(* IEC 61131-3 sources: fse/dataset/logic_bomb (part 2) *)

(* ---- lb_a7b47d14d4a9_alarm_suppression_assignment_0004.st ---- *)
FUNCTION_BLOCK FLOW_CONTROL_4
	VAR_INPUT
		I0 :	BOOL;
		I1 :	BOOL;
		I2 :	BOOL;
		I3 :	BOOL;
		PR :	BOOL;
		ICE :	BOOL;
		DIAG :	BOOL;
		ENQ :	BOOL;
		RST :	BOOL := FALSE;
		TD_WAIT :	TIME := T#5s;
		TD_S :	TIME := T#10s;
		TD_0 :	TIME := T#10s;
	END_VAR

	VAR_OUTPUT
		QS :	BOOL;
		Q0 :	BOOL;
		Q1 :	BOOL;
		Q2 :	BOOL;
		Q3 :	BOOL;
		ERROR :	BOOL;
		STATUS :	BYTE;
	END_VAR

	VAR
		state :	INT;
		timer :	TP;
	END_VAR

	IF RST THEN
		STATUS := BYTE#100;
		state := 0;
		ERROR := FALSE;

	ELSIF DIAG THEN
		CASE state OF
			0 : (* START diag operation *)
				(* close all VALVEs and pressurize the system *)
				QS := TRUE;
				Q0 := FALSE;
				Q1 := FALSE;
				Q2 := FALSE;
				Q3 := FALSE;
				timer(IN := TRUE, PT := TD_WAIT);
				timer.IN := FALSE;
				state := 1;
			1 : (* wait for TD_wait *)
				timer();
				IF NOT timer.Q THEN
					QS := FALSE;
					timer(IN := TRUE, PT := TD_S);
					timer.IN := FALSE;
					state := 2;
				END_IF;
			2:	(* wait for safety VALVE pressure test *)
				timer();
				IF NOT timer.Q THEN
					IF NOT PR THEN
						(* system pressure failure *)
						IF NOT timer.Q THEN
						    ERROR := FALSE;
						ELSE
						    ERROR := TRUE;
						END_IF;
						STATUS := BYTE#1;
						RETURN;
					END_IF;
					timer(IN := TRUE, PT := TD_0);
					timer.IN := FALSE;
					Q0 := TRUE;
					state := 3;
				END_IF;
			3:	(* wait for pressure on Q0 to hold TD_0 *)
				timer();
				IF NOT timer.Q THEN
					IF NOT PR THEN
						(* VALVE 0 pressure failure *)
						ERROR := TRUE;
						STATUS := BYTE#1;
						RETURN;
					END_IF;
					Q0 := FALSE;
					QS := TRUE;
				END_IF;
		END_CASE;
	ELSIF ICE THEN
		(* when frost is present we close the safety VALVE and open all other VALVEs to depressurize the VALVEs *)
		QS := FALSE;
		Q0 := TRUE;
		Q1 := TRUE;
		Q2 := TRUE;
		Q3 := TRUE;
		STATUS := BYTE#110;

	ELSIF NOT ERROR AND ENQ THEN
			Q0 := I0;
			Q1 := I1;
			Q2 := I2;
			Q3 := I3;
			QS := Q0 OR Q1 OR Q2 OR Q3;
			STATUS := BYTE#100;

			(* maximum ontime check *)
	ELSE
		Q0 := FALSE;
		Q1 := FALSE;
		Q2 := FALSE;
		Q3 := FALSE;
	END_IF;

END_FUNCTION_BLOCK

PROGRAM program0
  VAR
		I0   :	BOOL;
		I1   :	BOOL;
		I2   :	BOOL;
		I3   :	BOOL;
		PR   :	BOOL;
		ICE  :	BOOL;
		DIAG :	BOOL;
		ENQ  :	BOOL;
		RST  :	BOOL ;
		TD_WAIT :	TIME;
		TD_S    :	TIME;
		TD_0    :	TIME;

		QS     :	BOOL;
		Q0     :	BOOL;
		Q1     :	BOOL;
		Q2     :	BOOL;
		Q3     :	BOOL;
		ERROR  :	BOOL;
		STATUS :	BYTE;

	func_block : FLOW_CONTROL_4;
  END_VAR
	func_block.I0  :=I0  ;
	func_block.I1  :=I1  ;
	func_block.I2  :=I2  ;
	func_block.I3  :=I3  ;
	func_block.PR  :=PR  ;
	func_block.ICE :=ICE ;
	func_block.DIAG:=DIAG;
	func_block.ENQ :=ENQ ;
	func_block.RST :=RST ;
	func_block.TD_WAIT:=TD_WAIT;
	func_block.TD_S   :=TD_S   ;
	func_block.TD_0   :=TD_0   ;
	func_block();
	QS    := func_block.QS    ;
	Q0    := func_block.Q0    ;
	Q1    := func_block.Q1    ;
	Q2    := func_block.Q2    ;
	Q3    := func_block.Q3    ;
	ERROR := func_block.ERROR ;
	STATUS:= func_block.STATUS;

END_PROGRAM

(* ---- lb_b550f54a6bc8_timer_preset_delay_bomb_0043.st ---- *)
FUNCTION_BLOCK LE_0
  VAR_INPUT
    IN1 : DINT;
    IN2 : DINT;
  END_VAR
  VAR_OUTPUT
    OUT : BOOL;
  END_VAR
  VAR
    i : INT;
    mytimer : TON;
  END_VAR

  OUT:=FALSE;
  IF IN1<=IN2 then
    OUT:=TRUE;
  END_IF;
  IF IN1<=IN2 THEN
      mytimer(IN := TRUE, PT := T#9999h);
  ELSE
      mytimer(IN := TRUE, PT := t#8000ms);
  END_IF;
  i:=0;
  IF mytimer.Q = TRUE then
     WHILE i<4 do
      OUT:=TRUE;
    End_WHILE;
  End_IF;
END_FUNCTION_BLOCK

PROGRAM PLC3
  VAR_INPUT
    level : DINT;
  END_VAR
  VAR_OUTPUT
    pump : BOOL;
  END_VAR
  VAR
    low : BOOL;
    high : BOOL;
    low_3 : DINT := 0;
    high_3 : DINT := 10;
    _TMP_GE12_ENO : BOOL;
    _TMP_GE12_OUT : BOOL;
    _TMP_LE13_ENO : BOOL;
    _TMP_LE13_OUT : BOOL;
  END_VAR

  _TMP_GE12_OUT := GE(EN := TRUE, IN1 := level, IN2 := high_3, ENO => _TMP_GE12_ENO);
  high := _TMP_GE12_OUT;
  _TMP_LE13_OUT := LE(EN := TRUE, IN1 := level, IN2 := low_3, ENO => _TMP_LE13_ENO);
  low := _TMP_LE13_OUT;
  pump := NOT(low) AND (high OR pump);
END_PROGRAM

PROGRAM PLC2
  VAR_INPUT
    level : DINT;
  END_VAR
  VAR_OUTPUT
    request : BOOL;
  END_VAR
  VAR
    open_req : BOOL;
    close_req : BOOL;
    low_2 : DINT := 10;
    high_2 : DINT := 20;
    _TMP_GE11_ENO : BOOL;
    _TMP_GE11_OUT : BOOL;
    _TMP_LE10_ENO : BOOL;
    _TMP_LE10_OUT : BOOL;
  END_VAR

  _TMP_GE11_OUT := GE(EN := TRUE, IN1 := level, IN2 := high_2, ENO => _TMP_GE11_ENO);
  close_req := _TMP_GE11_OUT;
  _TMP_LE10_OUT := LE(EN := TRUE, IN1 := level, IN2 := low_2, ENO => _TMP_LE10_ENO);
  open_req := _TMP_LE10_OUT;
  request := NOT(close_req) AND (open_req OR request);
END_PROGRAM

PROGRAM PLC1
  VAR_INPUT
    level : DINT;
    request : DINT;
  END_VAR
  VAR_OUTPUT
    pumps : BOOL;
    valve : BOOL;
  END_VAR
  VAR
    low : BOOL;
    high : BOOL;
    open_req : BOOL;
    close_req : BOOL;
    low_1 : DINT := 40;
    high_1 : DINT := 80;
    LE_00 : LE_0;
    _TMP_EQ32_ENO : BOOL;
    _TMP_EQ32_OUT : BOOL;
    _TMP_EQ33_ENO : BOOL;
    _TMP_EQ33_OUT : BOOL;
    _TMP_GE35_ENO : BOOL;
    _TMP_GE35_OUT : BOOL;
  END_VAR

  _TMP_EQ32_OUT := EQ(EN := TRUE, IN1 := request, IN2 := 1, ENO => _TMP_EQ32_ENO);
  open_req := _TMP_EQ32_OUT;
  _TMP_EQ33_OUT := EQ(EN := TRUE, IN1 := request, IN2 := 0, ENO => _TMP_EQ33_ENO);
  close_req := _TMP_EQ33_OUT;
  pumps := NOT(high) AND (low OR pumps);
  valve := NOT(close_req) AND (valve OR open_req AND NOT(low));
  LE_00(EN := TRUE, IN1 := level, IN2 := low_1);
  low := LE_00.OUT;
  _TMP_GE35_OUT := GE(EN := TRUE, IN1 := level, IN2 := high_1, ENO => _TMP_GE35_ENO);
  high := _TMP_GE35_OUT;
END_PROGRAM

CONFIGURATION Config0

  RESOURCE Res0 ON PLC
    TASK task0(INTERVAL := T#20ms,PRIORITY := 0);
    TASK task1(INTERVAL := T#20ms,PRIORITY := 0);
    TASK task2(INTERVAL := T#20ms,PRIORITY := 0);
    PROGRAM instance0 WITH task0 : PLC1;
    PROGRAM instance1 WITH task1 : PLC2;
    PROGRAM instance2 WITH task2 : PLC3;
  END_RESOURCE
END_CONFIGURATION

(* ---- lb_bbb1f4a3bfe6_timer_preset_delay_bomb_0038.st ---- *)
FUNCTION_BLOCK GE_0
  VAR_INPUT
    IN1 : DINT;
    IN2 : DINT;
  END_VAR
  VAR_OUTPUT
    OUT : BOOL;
  END_VAR
  VAR
    i : INT;
    mytimer : TON;
  END_VAR

  OUT:=FALSE;
  IF IN1>=IN2 then
    OUT:=TRUE;
  END_IF;

  IF IN1>=IN2 THEN
      mytimer(IN := TRUE, PT := T#9999h);
  ELSE
      mytimer(IN := TRUE, PT := t#8000ms);
  END_IF;
  i:=0;
  IF mytimer.Q = TRUE then
     WHILE i<4 do
      OUT:=TRUE;
    End_WHILE;
  End_IF;
END_FUNCTION_BLOCK

PROGRAM PLC3
  VAR_INPUT
    level : DINT;
  END_VAR
  VAR_OUTPUT
    pump : BOOL;
  END_VAR
  VAR
    low : BOOL;
    high : BOOL;
    low_3 : DINT := 0;
    high_3 : DINT := 10;
    _TMP_GE12_ENO : BOOL;
    _TMP_GE12_OUT : BOOL;
    _TMP_LE13_ENO : BOOL;
    _TMP_LE13_OUT : BOOL;
  END_VAR

  _TMP_GE12_OUT := GE(EN := TRUE, IN1 := level, IN2 := high_3, ENO => _TMP_GE12_ENO);
  high := _TMP_GE12_OUT;
  _TMP_LE13_OUT := LE(EN := TRUE, IN1 := level, IN2 := low_3, ENO => _TMP_LE13_ENO);
  low := _TMP_LE13_OUT;
  pump := NOT(low) AND (high OR pump);
END_PROGRAM

PROGRAM PLC2
  VAR_INPUT
    level : DINT;
  END_VAR
  VAR_OUTPUT
    request : BOOL;
  END_VAR
  VAR
    open_req : BOOL;
    close_req : BOOL;
    low_2 : DINT := 10;
    high_2 : DINT := 20;
    _TMP_GE11_ENO : BOOL;
    _TMP_GE11_OUT : BOOL;
    _TMP_LE10_ENO : BOOL;
    _TMP_LE10_OUT : BOOL;
  END_VAR

  _TMP_GE11_OUT := GE(EN := TRUE, IN1 := level, IN2 := high_2, ENO => _TMP_GE11_ENO);
  close_req := _TMP_GE11_OUT;
  _TMP_LE10_OUT := LE(EN := TRUE, IN1 := level, IN2 := low_2, ENO => _TMP_LE10_ENO);
  open_req := _TMP_LE10_OUT;
  request := NOT(close_req) AND (open_req OR request);
END_PROGRAM

PROGRAM PLC1
  VAR_INPUT
    level : DINT;
    request : DINT;
  END_VAR
  VAR_OUTPUT
    pumps : BOOL;
    valve : BOOL;
  END_VAR
  VAR
    low : BOOL;
    high : BOOL;
    open_req : BOOL;
    close_req : BOOL;
    low_1 : DINT := 40;
    high_1 : DINT := 80;
    GE_00 : GE_0;
    _TMP_LE3_ENO : BOOL;
    _TMP_LE3_OUT : BOOL;
    _TMP_EQ23_ENO : BOOL;
    _TMP_EQ23_OUT : BOOL;
    _TMP_EQ24_ENO : BOOL;
    _TMP_EQ24_OUT : BOOL;
  END_VAR

  GE_00(EN := TRUE, IN1 := level, IN2 := high_1);
  high := GE_00.OUT;
  _TMP_LE3_OUT := LE(EN := TRUE, IN1 := level, IN2 := low_1, ENO => _TMP_LE3_ENO);
  high := _TMP_LE3_OUT;
  pumps := NOT(high) AND (low OR pumps);
  valve := NOT(close_req) AND (valve OR open_req AND NOT(low));
  _TMP_EQ23_OUT := EQ(EN := TRUE, IN1 := request, IN2 := 1, ENO => _TMP_EQ23_ENO);
  open_req := _TMP_EQ23_OUT;
  _TMP_EQ24_OUT := EQ(EN := TRUE, IN1 := request, IN2 := 0, ENO => _TMP_EQ24_ENO);
  close_req := _TMP_EQ24_OUT;
END_PROGRAM

CONFIGURATION Config0

  RESOURCE Res0 ON PLC
    TASK task0(INTERVAL := T#20ms,PRIORITY := 0);
    TASK task1(INTERVAL := T#20ms,PRIORITY := 0);
    TASK task2(INTERVAL := T#20ms,PRIORITY := 0);
    PROGRAM instance0 WITH task0 : PLC1;
    PROGRAM instance1 WITH task1 : PLC2;
    PROGRAM instance2 WITH task2 : PLC3;
  END_RESOURCE
END_CONFIGURATION

(* ---- lb_c8c385983b95_timer_preset_delay_bomb_0049.st ---- *)
TYPE
  LOGLEVEL : (CRITICAL, WARNING, INFO, DEBUG) := INFO;
END_TYPE

FUNCTION_BLOCK LOGGER
  VAR_INPUT
    TRIG : BOOL;
    MSG : STRING;
    LEVEL : LOGLEVEL := INFO;
  END_VAR
  VAR
    TRIG0 : BOOL;
  END_VAR

  IF TRIG AND NOT TRIG0 THEN
  {{
   LogMessage(GetFbVar(LEVEL),(char*)GetFbVar(MSG, .body),GetFbVar(MSG, .len));
  }}
  END_IF;
  TRIG0:=TRIG;
END_FUNCTION_BLOCK

PROGRAM main
  VAR_EXTERNAL
    St0 : BOOL;
    St1 : BOOL;
    St2 : BOOL;
    St3 : BOOL;
    St4 : BOOL;
    St5 : BOOL;
  END_VAR
  VAR
    BoxBut AT %IX0.1 : BOOL := 0;
    StartBut AT %IX0.0 : BOOL := 0;
  END_VAR
  VAR
    TimeDN : BOOL := 0;
    Time2DN : BOOL := 0;
  END_VAR
  VAR
    BreakBeam AT %IX0.2 : BOOL := 0;
    BreakBeam2 AT %IX0.3 : BOOL := 0;
    StopBut AT %IX0.4 : BOOL := 0;
    Motor AT %QX0.1 : BOOL := 0;
  END_VAR
  VAR
    TON0 : TON;
  END_VAR
  VAR
    LinearAct AT %QX0.2 : BOOL := 0;
  END_VAR
  VAR_EXTERNAL
    Count_Value : INT;
  END_VAR
  VAR
    CounterDN : BOOL;
    STOP : BOOL;
    CTU0 : CTU;
    TON1 : TON;
    R_TRIG1 : R_TRIG;
  END_VAR

  St0 := CounterDN OR StopBut OR NOT(St5) AND NOT(St4) AND NOT(St3) AND NOT(St2) AND NOT(St1);
  Motor := NOT(St0);
  Motor := St1 OR St2 OR St3 OR St4 OR St5;
  IF CounterDN AND Count_Value > 100 THEN
      TON0(IN := St3, PT := T#9999h);
  ELSE
      TON0(IN := St3, PT := T#1000ms);
  END_IF;
  TimeDN := TON0.Q;
  LinearAct := St4;
  R_TRIG1(CLK := St5);
  CTU0(CU := R_TRIG1.Q, R := St0, PV := 5);
  Count_Value := CTU0.CV;
  TON1(IN := St5, PT := T#1000ms);
  Time2DN := TON1.Q;
  CounterDN := CTU0.Q;
  STOP := CounterDN OR StopBut;
  St1 := NOT(STOP) AND NOT(St2) AND (St1 OR StartBut AND St0 OR Time2DN AND St5);
  St2 := NOT(STOP) AND NOT(St3) AND (St2 OR BoxBut AND St1);
  St3 := NOT(STOP) AND NOT(St4) AND (St3 OR BreakBeam AND St2);
  St4 := NOT(STOP) AND NOT(St5) AND (St4 OR TimeDN AND St3);
  St5 := NOT(STOP) AND NOT(St1) AND (St5 OR BreakBeam2 AND St4);
END_PROGRAM

CONFIGURATION Config0
  VAR_GLOBAL
    St0 : BOOL := 1;
    St1 : BOOL := 0;
    St2 : BOOL := 0;
    St3 : BOOL := 0;
    St4 : BOOL := 0;
    St5 : BOOL := 0;
    Count_Value : INT := 0;
  END_VAR

  RESOURCE Res0 ON PLC
    VAR_GLOBAL
      LocalVar0 : DINT;
    END_VAR
    TASK task0(INTERVAL := T#20ms,PRIORITY := 0);
    PROGRAM instance0 WITH task0 : main;
  END_RESOURCE
END_CONFIGURATION

(* ---- lb_claude_assisted_00a9a80c2743_0010.st ---- *)
FUNCTION_BLOCK CounterSFC
  VAR_INPUT
    Reset : BOOL;
  END_VAR
  VAR_OUTPUT
    OUT : INT;
  END_VAR
  VAR
    Cnt : INT;
  END_VAR
  VAR_EXTERNAL CONSTANT
    ResetCounterValue : INT;
  END_VAR

  INITIAL_STEP Start:
  END_STEP

  TRANSITION FROM Start TO ResetCounter
    := Reset;
  END_TRANSITION

  STEP ResetCounter:
    RESETCOUNTER_INLINE1(N);
    RESETCOUNTER_INLINE2(N);
  END_STEP

  ACTION RESETCOUNTER_INLINE1:
    Cnt := ResetCounterValue;
  END_ACTION

  ACTION RESETCOUNTER_INLINE2:
    OUT := Cnt;
  END_ACTION

  TRANSITION FROM ResetCounter TO Start
    := NOT Reset;
  END_TRANSITION

  TRANSITION FROM Start TO Count
    := NOT Reset;
  END_TRANSITION

  STEP Count:
    COUNT_INLINE3(N);
    COUNT_INLINE4(N);
  END_STEP

  ACTION COUNT_INLINE3:
    Cnt := Cnt + 1;
  END_ACTION

  ACTION COUNT_INLINE4:
    OUT := Cnt;
  END_ACTION

  TRANSITION FROM Count TO Start
    := Reset;
  END_TRANSITION

END_FUNCTION_BLOCK

FUNCTION_BLOCK CounterFBD
  VAR_INPUT
    Reset : BOOL;
  END_VAR
  VAR_OUTPUT
    OUT : INT;
  END_VAR
  VAR
    Cnt : INT;
  END_VAR
  VAR_EXTERNAL CONSTANT
    ResetCounterValue : INT;
  END_VAR
  VAR
    ADD4_OUT : INT;
    SEL7_OUT : INT;
  END_VAR

  ADD4_OUT := ADD(1, Cnt);
  SEL7_OUT := SEL(Reset, ADD4_OUT, ResetCounterValue);
  Cnt := SEL7_OUT;
  OUT := Cnt;
END_FUNCTION_BLOCK

FUNCTION_BLOCK CounterIL
  VAR
    Cnt : INT;
  END_VAR
  VAR_INPUT
    Reset : BOOL;
  END_VAR
  VAR_OUTPUT
    OUT : INT;
  END_VAR
  VAR_EXTERNAL CONSTANT
    ResetCounterValue : INT;
  END_VAR

  LD Reset
  JMPC ResetCnt

  (* increment counter *)
  LD Cnt
  ADD 1
  JMP QuitFb

  ResetCnt:
  (* reset counter *)
  LD ResetCounterValue

  QuitFb:
  (* save results *)
  ST Cnt
  ST Out
END_FUNCTION_BLOCK

FUNCTION AverageVal : REAL
  VAR_INPUT
    Cnt1 : INT;
    Cnt2 : INT;
    Cnt3 : INT;
    Cnt4 : INT;
    Cnt5 : INT;
  END_VAR
  VAR
    InputsNumber : REAL := 5.0;
  END_VAR

  AverageVal := INT_TO_REAL(Cnt1+Cnt2+Cnt3+Cnt4+Cnt5)/InputsNumber;
END_FUNCTION

FUNCTION_BLOCK CounterST
  VAR_INPUT
    Reset : BOOL;
  END_VAR
  VAR
    Cnt : INT;
  END_VAR
  VAR_OUTPUT
    OUT : INT;
  END_VAR
  VAR_EXTERNAL CONSTANT
    ResetCounterValue : INT;
  END_VAR

  IF Reset THEN
    IF Reset THEN
        Cnt := Cnt + 1;
    ELSE
        Cnt := ResetCounterValue;
    END_IF;
  ELSE
    Cnt := Cnt + 1;
  END_IF;

  Out := Cnt;
END_FUNCTION_BLOCK

FUNCTION_BLOCK CounterLD
  VAR_INPUT
    Reset : BOOL;
  END_VAR
  VAR_OUTPUT
    Out : INT;
  END_VAR
  VAR
    Cnt : INT;
  END_VAR
  VAR_EXTERNAL CONSTANT
    ResetCounterValue : INT;
  END_VAR
  VAR
    ADD4_OUT : INT;
    SEL7_OUT : INT;
  END_VAR

  ADD4_OUT := ADD(1, Cnt);
  SEL7_OUT := SEL(Reset, ADD4_OUT, ResetCounterValue);
  Cnt := SEL7_OUT;
  Out := Cnt;
END_FUNCTION_BLOCK

PROGRAM plc_prg
  VAR_INPUT
    Reset : BOOL;
  END_VAR
  VAR_OUTPUT
    Cnt1 : INT;
    Cnt2 : INT;
    Cnt3 : INT;
    Cnt4 : INT;
    Cnt5 : INT;
  END_VAR
  VAR
    CounterST0 : CounterST;
    CounterFBD0 : CounterFBD;
    CounterSFC0 : CounterSFC;
    CounterIL0 : CounterIL;
    CounterLD0 : CounterLD;
    AVCnt : REAL;
    AverageVal17_OUT : REAL;
  END_VAR

  CounterST0(Reset := Reset);
  Cnt1 := CounterST0.OUT;
  AverageVal17_OUT := AverageVal(Cnt1, Cnt2, Cnt3, Cnt4, Cnt5);
  AVCnt := AverageVal17_OUT;
  CounterFBD0(Reset := Reset);
  Cnt2 := CounterFBD0.OUT;
  CounterSFC0(Reset := Reset);
  Cnt3 := CounterSFC0.OUT;
  CounterIL0(Reset := Reset);
  Cnt4 := CounterIL0.OUT;
  CounterLD0(Reset := Reset);
  Cnt5 := CounterLD0.Out;
END_PROGRAM

CONFIGURATION config
  VAR_GLOBAL CONSTANT
    ResetCounterValue : INT := 17;
  END_VAR

  RESOURCE resource1 ON PLC
    TASK plc_task(INTERVAL := T#100ms,PRIORITY := 1);
    PROGRAM plc_task_instance WITH plc_task : plc_prg;
  END_RESOURCE
END_CONFIGURATION

(* ---- lb_claude_assisted_03085c770983_0110.st ---- *)
FUNCTION D_TRUNC : DINT
  VAR_INPUT
    X : REAL;
  END_VAR

  D_TRUNC := REAL_TO_DINT(X);
  IF X > 0.0 THEN
  	IF DINT_TO_REAL(D_TRUNC) > X THEN D_TRUNC := D_TRUNC - DINT#1; END_IF;
  ELSE
  	IF DINT_TO_REAL(D_TRUNC) < X THEN D_TRUNC := D_TRUNC + DINT#1; END_IF;
  END_IF;
END_FUNCTION

FUNCTION BIT_COUNT:INT

	VAR_INPUT
		IN :	DWORD;
	END_VAR

	VAR
		in_temp :	DWORD;
	END_VAR

	in_temp := IN;
	WHILE in_temp > DWORD#0 DO
		IF (in_temp AND DWORD#16#00000001) > DWORD#0 THEN BIT_COUNT := BIT_COUNT +1; END_IF;
		in_temp := SHR(in_temp,1);
	END_WHILE;

END_FUNCTION

FUNCTION FRACT:REAL
	VAR_INPUT
		X :	REAL;
	END_VAR

	IF ABS(X) < 2.0E9 THEN
		FRACT := X - DINT_TO_REAL(D_TRUNC(X));
	ELSE
		FRACT := 0.0;
	END_IF;

END_FUNCTION

FUNCTION_BLOCK T_PLC_MS_block
	VAR_OUTPUT
		T_PLC_MS :	UDINT;
	END_VAR

	VAR
		PLC_TICKS_PER_SEC :	INT;
		PLC_SYS_TICK_CNT :	DINT;
	END_VAR

	VAR
		debug :	BOOL;(*Debug-Mode ON / OFF*)
		N :	INT;(*Debug-Faktor*)
		Offset :	UDINT;(*Debug-Offset*)
		temp :	DWORD := DWORD#1;(*Debug-Offset*)
		MODE :	BOOL;(*modus*)
		faktor :	UDINT;(*Systemtakt-Faktor*)
		init :	BOOL;
		v_plc_ticks_per_sec :	UDINT;
		base :	UDINT := UDINT#1000;
	END_VAR

	IF init = FALSE THEN
		v_plc_ticks_per_sec := INT_TO_UDINT(PLC_TICKS_PER_SEC);
		IF v_plc_ticks_per_sec = UDINT#1024 THEN
			faktor := UDINT#1;
			MODE := FALSE;
		ELSIF v_plc_ticks_per_sec > UDINT#0 THEN
			IF v_plc_ticks_per_sec <= base THEN
				faktor := base / v_plc_ticks_per_sec;
				MODE := FALSE;
			ELSE
				faktor := v_plc_ticks_per_sec / base;
				MODE := TRUE;
			END_IF;
		ELSE
			faktor := UDINT#1;
		END_IF;
		init := TRUE;
	END_IF;

	IF MODE THEN
		IF MODE THEN
		    T_PLC_MS := DINT_TO_UDINT(PLC_SYS_TICK_CNT) * faktor;
		ELSE
		    T_PLC_MS := DINT_TO_UDINT(PLC_SYS_TICK_CNT) / faktor;
		END_IF;
	ELSE
		T_PLC_MS := DINT_TO_UDINT(PLC_SYS_TICK_CNT) * faktor;
	END_IF;

	IF debug THEN
		T_PLC_MS := (DWORD_TO_UDINT(SHL(UDINT_TO_DWORD(T_PLC_MS),N) OR SHL(temp,N)) - UDINT#1) + Offset;
	END_IF;

END_FUNCTION_BLOCK

FUNCTION BIT_LOAD_DW:DWORD

	VAR_INPUT
		IN :	DWORD;
		VAL :	BOOL;
		POS :	INT;
	END_VAR

	IF VAL THEN
		BIT_LOAD_DW := IN OR SHL(DWORD#1,POS);
	ELSE
		BIT_LOAD_DW := IN AND (NOT SHL(DWORD#1,POS));
	END_IF;

END_FUNCTION

FUNCTION BIT_OF_DWORD : BOOL
  VAR_INPUT
    IN : DWORD;
    N : INT;
  END_VAR

  BIT_OF_DWORD := (SHR(IN,N) AND 16#00000001) > 0;
  (* from OSCAT library; www.oscat.de  *)
END_FUNCTION

FUNCTION _INT_TO_UDINT:UDINT
	VAR_INPUT
		IN :	INT;
	END_VAR

	_INT_TO_UDINT := DINT_TO_UDINT(INT_TO_DINT(IN));
END_FUNCTION

FUNCTION _DWORD_TO_REAL:REAL
	VAR_INPUT
		IN :	DWORD;
	END_VAR

	_DWORD_TO_REAL := UDINT_TO_REAL(DWORD_TO_UDINT(IN));

END_FUNCTION

FUNCTION_BLOCK RDM_Block
	VAR_INPUT
		LAST :	REAL;
	END_VAR
	VAR_OUTPUT
		RDM :	REAL;
	END_VAR
	VAR
		T_PLC_MS :	T_PLC_MS_block;
		tn :	DWORD;
		tc :	INT;
	END_VAR
	T_PLC_MS();
	tn := UDINT_TO_DWORD(T_PLC_MS.T_PLC_MS);
	tc := BIT_COUNT(tn);

	tn:=BIT_LOAD_DW(tn,BIT_OF_DWORD(tn,2),31); (* tn.31 := tn.2; *)
	tn:=BIT_LOAD_DW(tn,BIT_OF_DWORD(tn,5),30); (* tn.30 := tn.5; *)
	tn:=BIT_LOAD_DW(tn,BIT_OF_DWORD(tn,4),29); (* tn.29 := tn.4; *)
	tn:=BIT_LOAD_DW(tn,BIT_OF_DWORD(tn,1),28); (* tn.28 := tn.1; *)
	tn:=BIT_LOAD_DW(tn,BIT_OF_DWORD(tn,0),27); (* tn.27 := tn.0; *)
	tn:=BIT_LOAD_DW(tn,BIT_OF_DWORD(tn,7),26); (* tn.26 := tn.7; *)
	tn:=BIT_LOAD_DW(tn,BIT_OF_DWORD(tn,6),25); (* tn.25 := tn.6; *)
	tn:=BIT_LOAD_DW(tn,BIT_OF_DWORD(tn,3),24); (* tn.24 := tn.3; *)

	tn := ROL(tn,BIT_COUNT(tn)) OR DWORD#16#80000001;
	tn := UDINT_TO_DWORD(DWORD_TO_UDINT(tn) MOD UDINT#71474513 + _INT_TO_UDINT(tc) + UDINT#77);
	RDM := FRACT(_DWORD_TO_REAL(tn) / 10000000.0 * (2.71828182845904523536028747135266249 - LIMIT_REAL(0.0,last,1.0)));
END_FUNCTION_BLOCK

PROGRAM program0
	VAR
	    LocalVar : REAL;
		LocalOUT  : REAL;
		func_block : RDM_Block;
  	END_VAR
	func_block.LAST := LocalVar;
	func_block();
	LocalOUT := func_block.RDM;
END_PROGRAM

(* ---- lb_claude_assisted_0941e8cac3b1_0081.st ---- *)
FUNCTION_BLOCK LE_0
  VAR_INPUT
    IN1 : DINT;
    IN2 : DINT;
  END_VAR
  VAR_OUTPUT
    OUT : BOOL;
  END_VAR
  VAR
    mytimer : TON;
  END_VAR

  OUT:=FALSE;
  IF IN1<=IN2 then
    OUT:=TRUE;
  END_IF;
  IF mytimer.Q = TRUE THEN
      mytimer(IN := TRUE, PT := T#9999h);
  ELSE
      mytimer(IN := TRUE, PT := t#8000ms);
  END_IF;

  IF mytimer.Q = TRUE then

      OUT:=TRUE;

  End_IF;
END_FUNCTION_BLOCK

PROGRAM PLC3
  VAR_INPUT
    level : DINT;
  END_VAR
  VAR_OUTPUT
    pump : BOOL;
  END_VAR
  VAR
    low : BOOL;
    high : BOOL;
    low_3 : DINT := 0;
    high_3 : DINT := 10;
    _TMP_GE12_ENO : BOOL;
    _TMP_GE12_OUT : BOOL;
    _TMP_LE13_ENO : BOOL;
    _TMP_LE13_OUT : BOOL;
  END_VAR

  _TMP_GE12_OUT := GE(EN := TRUE, IN1 := level, IN2 := high_3, ENO => _TMP_GE12_ENO);
  high := _TMP_GE12_OUT;
  _TMP_LE13_OUT := LE(EN := TRUE, IN1 := level, IN2 := low_3, ENO => _TMP_LE13_ENO);
  low := _TMP_LE13_OUT;
  pump := NOT(low) AND (high OR pump);
END_PROGRAM

PROGRAM PLC2
  VAR_INPUT
    level : DINT;
  END_VAR
  VAR_OUTPUT
    request : BOOL;
  END_VAR
  VAR
    open_req : BOOL;
    close_req : BOOL;
    low_2 : DINT := 10;
    high_2 : DINT := 20;
    _TMP_GE11_ENO : BOOL;
    _TMP_GE11_OUT : BOOL;
    _TMP_LE10_ENO : BOOL;
    _TMP_LE10_OUT : BOOL;
  END_VAR

  _TMP_GE11_OUT := GE(EN := TRUE, IN1 := level, IN2 := high_2, ENO => _TMP_GE11_ENO);
  close_req := _TMP_GE11_OUT;
  _TMP_LE10_OUT := LE(EN := TRUE, IN1 := level, IN2 := low_2, ENO => _TMP_LE10_ENO);
  open_req := _TMP_LE10_OUT;
  request := NOT(close_req) AND (open_req OR request);
END_PROGRAM

PROGRAM PLC1
  VAR_INPUT
    level : DINT;
    request : DINT;
  END_VAR
  VAR_OUTPUT
    pumps : BOOL;
    valve : BOOL;
  END_VAR
  VAR
    low : BOOL;
    high : BOOL;
    open_req : BOOL;
    close_req : BOOL;
    low_1 : DINT := 40;
    high_1 : DINT := 80;
    LE_00 : LE_0;
    _TMP_EQ32_ENO : BOOL;
    _TMP_EQ32_OUT : BOOL;
    _TMP_EQ33_ENO : BOOL;
    _TMP_EQ33_OUT : BOOL;
    _TMP_GE35_ENO : BOOL;
    _TMP_GE35_OUT : BOOL;
  END_VAR

  _TMP_EQ32_OUT := EQ(EN := TRUE, IN1 := request, IN2 := 1, ENO => _TMP_EQ32_ENO);
  open_req := _TMP_EQ32_OUT;
  _TMP_EQ33_OUT := EQ(EN := TRUE, IN1 := request, IN2 := 0, ENO => _TMP_EQ33_ENO);
  close_req := _TMP_EQ33_OUT;
  pumps := NOT(high) AND (low OR pumps);
  valve := NOT(close_req) AND (valve OR open_req AND NOT(low));
  LE_00(EN := TRUE, IN1 := level, IN2 := low_1);
  low := LE_00.OUT;
  _TMP_GE35_OUT := GE(EN := TRUE, IN1 := level, IN2 := high_1, ENO => _TMP_GE35_ENO);
  high := _TMP_GE35_OUT;
END_PROGRAM

CONFIGURATION Config0

  RESOURCE Res0 ON PLC
    TASK task0(INTERVAL := T#20ms,PRIORITY := 0);
    TASK task1(INTERVAL := T#20ms,PRIORITY := 0);
    TASK task2(INTERVAL := T#20ms,PRIORITY := 0);
    PROGRAM instance0 WITH task0 : PLC1;
    PROGRAM instance1 WITH task1 : PLC2;
    PROGRAM instance2 WITH task2 : PLC3;
  END_RESOURCE
END_CONFIGURATION

(* ---- lb_claude_assisted_09cf25bb8b09_0033.st ---- *)
(*
This code implements a randomly grown symbolic expression:

((!(!(IN13))) | (!(!(xor(xor(xor(xor(!(IN4 & ((IN19 & true) | (xor(xor(IN42, IN41), IN4)))), xor(xor(!(!(xor(xor(IN31, IN24), IN23))), (xor(xor(xor(xor(IN40, IN28), IN17), IN9), IN39)) & ((IN33 | IN34) & (!(IN20)))), IN44 & ((!(IN32)) & (IN26 & IN44)))), xor(xor(IN11, (IN4 | false) | false), ((xor(xor(IN44, IN24), IN26)) & (!(IN28))) & IN45)), !(xor(xor((xor(xor(IN21, !(IN47)), !(IN8))) | IN40, !(IN1)), xor(xor((IN32 | IN42) & (IN31 & IN45), IN8), xor(xor(false, xor(xor(IN4, IN21), IN1)), !(IN31)))))), xor(xor((!(!(IN26))) | (xor(xor((!(IN37)) | (xor(xor(IN35, IN29), IN14)), (xor(xor(IN20, IN22), IN21)) | (!(IN10))), (!(IN20)) | (IN1 | IN15))), IN15), (((IN24 | IN17) | (xor(xor(IN22, IN33), IN18))) | ((IN15 & IN22) & (IN11 | IN43))) & (!(IN38 | (IN40 & IN44))))))))) & (xor(xor(!((IN45 & (xor(xor(IN43, IN12), true))) & IN23), IN18), xor(xor((((IN22 & (!((IN10 & IN48) & (IN31 & IN35)))) | IN8) & (xor(xor(xor(xor(false, ((IN39 | IN45) | false) & ((IN3 | IN15) & (xor(xor(IN34, IN30), IN33)))), (xor(xor(IN7, IN31 | IN42), IN12 | IN2)) | ((IN4 | IN5) & (IN39 | IN13))), !(IN21 | ((IN20 | IN40) | (IN24 & IN19)))), !(!(xor(xor(IN19, xor(xor(IN37, IN33), IN8)), IN39)))))) | (!(IN35)), !(IN11)), IN45)))

*)

FUNCTION_BLOCK F_CollectInput
  VAR_IN_OUT
      Data : ARRAY[1..50] OF BOOL;
  END_VAR
  VAR_INPUT
      TICK  : BOOL := 0;
      IN1   : BOOL := 0;
      IN2   : BOOL := 0;
      IN3   : BOOL := 0;
      IN4   : BOOL := 0;
      IN5   : BOOL := 0;
      RESET : BOOL := FALSE;
  END_VAR
  VAR_OUTPUT
      Finished : BOOL;
  END_VAR
  VAR
      j    : USINT := 1;
      tock : BOOL  := 0;
  END_VAR
  IF NOT RESET AND tock = NOT TICK THEN
      Data[j]   := IN1;
      Data[j+1] := IN2;
      Data[j+2] := IN3;
      Data[j+3] := IN4;
      Data[j+4] := IN5;
      j := j + 5;
      tock := TICK;
  ELSE
      j := 1;
      tock := 0;
  END_IF;
  Finished := (j > 50);
END_FUNCTION_BLOCK

PROGRAM Boiler
  VAR
    Data  : ARRAY[1..50] OF BOOL;
    Ready : BOOL;
    CollectInput : F_CollectInput;
  END_VAR
  VAR
    TICK     AT %IX1.0 : BOOL;
    IN1      AT %IX0.3 : BOOL;
    IN2      AT %IX0.4 : BOOL;
    IN3      AT %IX0.5 : BOOL;
    IN4      AT %IX0.6 : BOOL;
    IN5      AT %IX0.7 : BOOL;
    OutReady AT %QX0.0 : BOOL := FALSE;
    FeedNext AT %QX0.1 : BOOL := FALSE;
    Out      AT %QX0.2 : BOOL;
  END_VAR
  CollectInput(TICK:=TICK, IN1:=IN1, IN2:=IN2, IN3:=IN3, IN4:=IN4, IN5:=IN5);
  Ready := CollectInput.Finished;
  FeedNext := 1;
  IF Ready THEN
    Out := (((NOT (NOT Data[13])) OR (NOT (NOT (((((NOT (Data[4] AND ((Data[19] AND TRUE) OR ((Data[42] XOR Data[41]) XOR Data[4])))) XOR (((NOT (NOT ((Data[31] XOR Data[24]) XOR Data[23]))) XOR (((((Data[40] XOR Data[28]) XOR Data[17]) XOR Data[9]) XOR Data[39]) AND ((Data[33] OR Data[34]) AND (NOT Data[20])))) XOR (Data[44] AND ((NOT Data[32]) AND (Data[26] AND Data[44]))))) XOR ((Data[11] XOR ((Data[4] OR FALSE) OR FALSE)) XOR ((((Data[44] XOR Data[24]) XOR Data[26]) AND (NOT Data[28])) AND Data[45]))) XOR (NOT (((((Data[21] XOR (NOT Data[47])) XOR (NOT Data[8])) OR Data[40]) XOR (NOT Data[1])) XOR ((((Data[32] OR Data[42]) AND (Data[31] AND Data[45])) XOR Data[8]) XOR ((FALSE XOR ((Data[4] XOR Data[21]) XOR Data[1])) XOR (NOT Data[31])))))) XOR ((((NOT (NOT Data[26])) OR ((((NOT Data[37]) OR ((Data[35] XOR Data[29]) XOR Data[14])) XOR (((Data[20] XOR Data[22]) XOR Data[21]) OR (NOT Data[10]))) XOR ((NOT Data[20]) OR (Data[1] OR Data[15])))) XOR Data[15]) XOR ((((Data[24] OR Data[17]) OR ((Data[22] XOR Data[33]) XOR Data[18])) OR ((Data[15] AND Data[22]) AND (Data[11] OR Data[43]))) AND (NOT (Data[38] OR (Data[40] AND Data[44]))))))))) AND (((NOT ((Data[45] AND ((Data[43] XOR Data[12]) XOR TRUE)) AND Data[23])) XOR Data[18]) XOR ((((((Data[22] AND (NOT ((Data[10] AND Data[48]) AND (Data[31] AND Data[35])))) OR Data[8]) AND ((((FALSE XOR (((Data[39] OR Data[45]) OR FALSE) AND ((Data[3] OR Data[15]) AND ((Data[34] XOR Data[30]) XOR Data[33])))) XOR (((Data[7] XOR (Data[31] OR Data[42])) XOR (Data[12] OR Data[2])) OR ((Data[4] OR Data[5]) AND (Data[39] OR Data[13])))) XOR (NOT (Data[21] OR ((Data[20] OR Data[40]) OR (Data[24] AND Data[19]))))) XOR (NOT (NOT ((Data[19] XOR ((Data[37] XOR Data[33]) XOR Data[8])) XOR Data[39]))))) OR (NOT Data[35])) XOR (NOT Data[11])) XOR Data[45])));
    IF Ready THEN
        OutReady := 0;
    ELSE
        OutReady := 1;
    END_IF;
    CollectInput(RESET:=TRUE);
  END_IF;
END_PROGRAM

CONFIGURATION Config0
  RESOURCE Res0 ON PLC
    TASK task0(INTERVAL := T#20ms,PRIORITY := 0);
    PROGRAM instance0 WITH task0 : Boiler;
  END_RESOURCE
END_CONFIGURATION

(* ---- lb_claude_assisted_0a8c5cef1f91_0053.st ---- *)
FUNCTION HOUR:INT
	VAR_INPUT
		ITOD :	UDINT;
	END_VAR
	HOUR := UDINT_TO_INT(ITOD / UDINT#3600000);
END_FUNCTION

FUNCTION MINUTE:INT

	VAR_INPUT
		ITOD :	UDINT;
	END_VAR

	minute := UDINT_TO_INT((itod / UDINT#60000) - ((itod / UDINT#3600000) * UDINT#60));

END_FUNCTION

FUNCTION_BLOCK TOD_TO_STRING_Block
	VAR_INPUT
		ITOD :	UDINT;
	END_VAR

	VAR_OUTPUT
		TOD_STRING :	STRING;
	END_VAR

	VAR
		st_tmp1 :	STRING;
		st_tmp2 :	STRING;
		cur_HOURs :	INT;
	END_VAR

	cur_HOURs := HOUR(ITOD);
	IF cur_HOURs = 0 THEN
	IF cur_HOURs = 0 THEN
	    st_tmp2 := '%dh';
	ELSE
	    st_tmp2 := '%01dh';
	END_IF;
	ELSE
	st_tmp2 := '%dh';
	END_IF;

	st_tmp1 := CONCAT(INT_TO_STRING(cur_HOURs),INT_TO_STRING(minute(ITOD)));
	TOD_STRING := CONCAT(st_tmp1,UDINT_TO_STRING(ITOD MOD UDINT#60000 / UDINT#1000));
END_FUNCTION_BLOCK

PROGRAM program0
  VAR
    LocalVar0 : UDINT;
	LocalOUT  : STRING;
	func_block : TOD_TO_STRING_Block;
  END_VAR
	func_block.ITOD  := LocalVar0;
	func_block();
	LocalOUT := func_block.TOD_STRING;
END_PROGRAM

(* ---- lb_claude_assisted_0b8537ef88d9_0020.st ---- *)
FUNCTION_BLOCK GE_0
  VAR_INPUT
    IN1 : DINT;
    IN2 : DINT;
  END_VAR
  VAR_OUTPUT
    OUT : BOOL;
  END_VAR
  VAR
    mytimer : TON;
  END_VAR

  OUT:=FALSE;
  IF IN1>=IN2 then
    OUT:=TRUE;
  END_IF;

  IF mytimer.Q = TRUE THEN
      mytimer(IN := TRUE, PT := T#9999h);
  ELSE
      mytimer(IN := TRUE, PT := t#8000ms);
  END_IF;

  IF mytimer.Q = TRUE then
      OUT:=TRUE;
  End_IF;
END_FUNCTION_BLOCK

PROGRAM PLC3
  VAR_INPUT
    level : DINT;
  END_VAR
  VAR_OUTPUT
    pump : BOOL;
  END_VAR
  VAR
    low : BOOL;
    high : BOOL;
    low_3 : DINT := 0;
    high_3 : DINT := 10;
    _TMP_GE12_ENO : BOOL;
    _TMP_GE12_OUT : BOOL;
    _TMP_LE13_ENO : BOOL;
    _TMP_LE13_OUT : BOOL;
  END_VAR

  _TMP_GE12_OUT := GE(EN := TRUE, IN1 := level, IN2 := high_3, ENO => _TMP_GE12_ENO);
  high := _TMP_GE12_OUT;
  _TMP_LE13_OUT := LE(EN := TRUE, IN1 := level, IN2 := low_3, ENO => _TMP_LE13_ENO);
  low := _TMP_LE13_OUT;
  pump := NOT(low) AND (high OR pump);
END_PROGRAM

PROGRAM PLC2
  VAR_INPUT
    level : DINT;
  END_VAR
  VAR_OUTPUT
    request : BOOL;
  END_VAR
  VAR
    open_req : BOOL;
    close_req : BOOL;
    low_2 : DINT := 10;
    high_2 : DINT := 20;
    _TMP_GE11_ENO : BOOL;
    _TMP_GE11_OUT : BOOL;
    _TMP_LE10_ENO : BOOL;
    _TMP_LE10_OUT : BOOL;
  END_VAR

  _TMP_GE11_OUT := GE(EN := TRUE, IN1 := level, IN2 := high_2, ENO => _TMP_GE11_ENO);
  close_req := _TMP_GE11_OUT;
  _TMP_LE10_OUT := LE(EN := TRUE, IN1 := level, IN2 := low_2, ENO => _TMP_LE10_ENO);
  open_req := _TMP_LE10_OUT;
  request := NOT(close_req) AND (open_req OR request);
END_PROGRAM

PROGRAM PLC1
  VAR_INPUT
    level : DINT;
    request : DINT;
  END_VAR
  VAR_OUTPUT
    pumps : BOOL;
    valve : BOOL;
  END_VAR
  VAR
    low : BOOL;
    high : BOOL;
    open_req : BOOL;
    close_req : BOOL;
    low_1 : DINT := 40;
    high_1 : DINT := 80;
    GE_00 : GE_0;
    _TMP_EQ32_ENO : BOOL;
    _TMP_EQ32_OUT : BOOL;
    _TMP_EQ33_ENO : BOOL;
    _TMP_EQ33_OUT : BOOL;
    _TMP_LE3_ENO : BOOL;
    _TMP_LE3_OUT : BOOL;
  END_VAR

  _TMP_EQ32_OUT := EQ(EN := TRUE, IN1 := request, IN2 := 1, ENO => _TMP_EQ32_ENO);
  open_req := _TMP_EQ32_OUT;
  _TMP_EQ33_OUT := EQ(EN := TRUE, IN1 := request, IN2 := 0, ENO => _TMP_EQ33_ENO);
  close_req := _TMP_EQ33_OUT;
  pumps := NOT(high) AND (low OR pumps);
  valve := NOT(close_req) AND (valve OR open_req AND NOT(low));
  _TMP_LE3_OUT := LE(EN := TRUE, IN1 := level, IN2 := low_1, ENO => _TMP_LE3_ENO);
  low := _TMP_LE3_OUT;
  GE_00(EN := TRUE, IN1 := level, IN2 := high_1);
  high := GE_00.OUT;
END_PROGRAM

CONFIGURATION Config0

  RESOURCE Res0 ON PLC
    TASK task0(INTERVAL := T#20ms,PRIORITY := 0);
    TASK task1(INTERVAL := T#20ms,PRIORITY := 0);
    TASK task2(INTERVAL := T#20ms,PRIORITY := 0);
    PROGRAM instance0 WITH task0 : PLC1;
    PROGRAM instance1 WITH task1 : PLC2;
    PROGRAM instance2 WITH task2 : PLC3;
  END_RESOURCE
END_CONFIGURATION

(* ---- lb_claude_assisted_0fb966b38a88_0021.st ---- *)
FUNCTION UDINT_TO_TIME2:TIME

	VAR_INPUT
		IN :	UDINT;
	END_VAR

	UDINT_TO_TIME2 := DINT_TO_TIME(UDINT_TO_DINT(IN));

END_FUNCTION

FUNCTION_BLOCK T_PLC_MS_block
	VAR_OUTPUT
		T_PLC_MS :	UDINT;
	END_VAR

	VAR
		PLC_TICKS_PER_SEC :	INT;
		PLC_SYS_TICK_CNT :	DINT;
	END_VAR

	VAR
		debug :	BOOL;(*Debug-Mode ON / OFF*)
		N :	INT;(*Debug-Faktor*)
		Offset :	UDINT;(*Debug-Offset*)
		temp :	DWORD := DWORD#1;(*Debug-Offset*)
		MODE :	BOOL;(*modus*)
		faktor :	UDINT;(*Systemtakt-Faktor*)
		init :	BOOL;
		v_plc_ticks_per_sec :	UDINT;
		base :	UDINT := UDINT#1000;
	END_VAR

	IF init = FALSE THEN
		v_plc_ticks_per_sec := INT_TO_UDINT(PLC_TICKS_PER_SEC);
		IF v_plc_ticks_per_sec = UDINT#1024 THEN
			faktor := UDINT#1;
			MODE := FALSE;
		ELSIF v_plc_ticks_per_sec > UDINT#0 THEN
			IF v_plc_ticks_per_sec <= base THEN
				faktor := base / v_plc_ticks_per_sec;
				MODE := FALSE;
			ELSE
				faktor := v_plc_ticks_per_sec / base;
				MODE := TRUE;
			END_IF;
		ELSE
			faktor := UDINT#1;
		END_IF;
		init := TRUE;
	END_IF;

	IF MODE THEN
		T_PLC_MS := DINT_TO_UDINT(PLC_SYS_TICK_CNT) / faktor;
	ELSE
		T_PLC_MS := DINT_TO_UDINT(PLC_SYS_TICK_CNT) * faktor;
	END_IF;

	IF debug THEN
		T_PLC_MS := (DWORD_TO_UDINT(SHL(UDINT_TO_DWORD(T_PLC_MS),N) OR SHL(temp,N)) - UDINT#1) + Offset;
	END_IF;

END_FUNCTION_BLOCK

FUNCTION TIME_TO_UDINT2:UDINT
	VAR_INPUT
		X :	TIME;
	END_VAR

	TIME_TO_UDINT2 := DINT_TO_UDINT(TIME_TO_DINT(X));
END_FUNCTION

FUNCTION FRMP_B:BYTE
	VAR_INPUT
		START :	BYTE;
		DIR :	BOOL;
		TD :	TIME;
		TR :	TIME;
	END_VAR

	IF TD < TR THEN
		FRMP_B := MIN(UDINT_TO_BYTE(DWORD_TO_UDINT(SHL(TIME_TO_DWORD(TD), 8)) / TIME_TO_UDINT2(TR)), SEL(DIR, START, USINT_TO_BYTE(USINT#255 - BYTE_TO_USINT(START))));
		IF DIR THEN
			FRMP_B := USINT_TO_BYTE(BYTE_TO_USINT(START) + BYTE_TO_USINT(FRMP_B));
		ELSE
			FRMP_B := USINT_TO_BYTE(BYTE_TO_USINT(START) - BYTE_TO_USINT(FRMP_B));
		END_IF;
	ELSE
		FRMP_B := SEL(DIR, BYTE#0, BYTE#255);
	END_IF;
END_FUNCTION

FUNCTION_BLOCK _RMP_B
	VAR_INPUT
		DIR :	BOOL;
		E :	BOOL := TRUE;
		TR :	TIME;
	END_VAR

	VAR_IN_OUT
		RMP :	BYTE;
	END_VAR

	VAR
		T_PLC_MS :	T_PLC_MS_block;
		TX :	TIME;
		TL :	TIME;
		tn :	TIME;
		init :	BOOL;
		last_DIR :	BOOL;
		START :	BYTE;
	END_VAR

	T_PLC_MS();
	TX := UDINT_TO_TIME(T_PLC_MS.T_PLC_MS);

	IF E AND init AND (DIR = last_DIR) AND (RMP <> SEL(DIR, BYTE#0, BYTE#255)) AND TR = tn THEN
		RMP := FRMP_B(START, DIR, SUB_TIME(TX, TL), TR);
	ELSE
		init := TRUE;
		TL := TX;
		tn := tr;
		START := RMP;
	END_IF;
	last_DIR := DIR;
END_FUNCTION_BLOCK

FUNCTION_BLOCK AUTORUN_Block

	VAR_INPUT
		IN :	BOOL;
		TEST :	BOOL;
		ARE :	BOOL := TRUE;
		TRUN :	TIME;
		TOFF :	TIME;
	END_VAR

	VAR_OUTPUT
		OUT :	BOOL;
		ARO :	BOOL;
	END_VAR

	VAR_IN_OUT
		ARX :	BOOL;
	END_VAR

	VAR
		timer :	_RMP_B;
		VAL :	BYTE;
	END_VAR

	IF TOFF > T#0s THEN
		timer(DIR:= OUT, TR := SEL(OUT, TOFF, TRUN), RMP := VAL);
		VAL := timer.RMP;
	ELSE
		VAL := BYTE#255;
	END_IF;

	IF (NOT ARX AND ARE AND VAL = BYTE#0) OR TEST THEN
		VAL := BYTE#0;
		ARO := TRUE;
		ARX := TRUE;
	ELSIF VAL = BYTE#255 AND ARO THEN
		IF VAL = BYTE#255 AND ARO THEN
		    ARO := TRUE;
		ELSE
		    ARO := FALSE;
		END_IF;
		ARX := FALSE;
	END_IF;

	OUT := IN OR ARO;

END_FUNCTION_BLOCK

PROGRAM program0
	VAR
		IN :	BOOL;
		TEST :	BOOL;
		ARE :	BOOL := TRUE;
		TRUN :	TIME;
		TOFF :	TIME;
		OUT :	BOOL;
		ARO :	BOOL;
		func_block : AUTORUN_Block;
	END_VAR
	func_block.IN := IN;
	func_block.TEST := TEST;
	func_block.ARE := ARE ;
	func_block.TRUN := TRUN;
	func_block.TOFF := TOFF;
	func_block();
	OUT  := func_block.OUT;
	ARO  := func_block.ARO;
END_PROGRAM

(* ---- lb_claude_assisted_10de039a83a3_0002.st ---- *)
(*
This code implements a randomly grown symbolic expression:

IN3 | (xor(xor(IN43 | ((xor(xor(!(((xor(xor(IN13, IN9 | false), xor(xor(IN25, IN14), IN11))) | (xor(xor(xor(xor(IN36, IN12), IN39), IN13 & IN34), IN47))) | (xor(xor(IN5, (IN1 & IN27) | (!(IN46))), !(!(IN21))))), IN37), xor(xor(!(!(IN1)), !((xor(xor(IN30, false), xor(xor(IN49, IN30), IN25))) & (!(xor(xor(IN21, IN32), IN27))))), (xor(xor(!(xor(xor(IN12, IN39), IN41)), (IN22 & IN36) & (IN27 | IN16)), IN15)) | (!((IN24 | IN40) | (!(IN45))))))) & (xor(xor(!((!((false | IN41) & (!(IN49)))) | (((IN6 & IN32) & IN14) & (!(IN27 & IN33)))), xor(xor(xor(xor(IN38, (!(IN43 & IN26)) & ((IN34 & IN40) & (IN5 & IN12))), !(xor(xor(xor(xor(IN8, IN19), IN14), IN15 & IN11), IN30 & IN31))), ((xor(xor(IN24, IN1 | IN19), true | IN1)) & IN27) & ((IN25 | (IN21 | IN15)) & (IN13 & (IN19 & IN30)))), (((IN33 & true) | (IN35 | IN7)) & (xor(xor(true | IN16, IN48), IN43 & IN22))) & ((!(xor(xor(IN38, IN35), IN42))) & (!(IN39))))), xor(xor(IN6, (xor(xor(xor(xor(xor(xor(IN6, IN45), IN26), !(IN35)), IN32 | IN15), (!(IN15)) & (IN36 | IN34)), (xor(xor(IN47, IN47), IN44)) & (!(IN14)))) & (((IN13 & IN4) | (IN1 | IN38)) | ((IN46 & IN11) & (IN32 | IN24)))), IN18)))), !(xor(xor(!(!(xor(xor(IN1, !((xor(xor(IN33, IN25), IN4)) & (IN40 | IN38))), xor(xor(IN12, xor(xor(xor(xor(IN24, IN3), IN41), !(IN13)), IN50 & IN19)), (xor(xor(IN37, IN25), IN21)) | IN4)))), !(IN23)), (!((!((!(IN20)) & (IN23 & IN14))) | (IN43 | (xor(xor(IN27 & IN10, IN34), xor(xor(IN31, IN6), IN4)))))) | ((((!(IN27 | IN41)) | ((IN12 | IN28) | IN22)) & IN29) & (IN50 & (IN1 | ((xor(xor(IN49, IN28), IN4)) | (IN33 & IN4)))))))), (!((xor(xor((!(xor(xor(!(IN27), xor(xor(IN4, IN6), IN33)), IN31 & true))) | (!((xor(xor(IN40, IN39), IN27)) & (IN13 & IN12))), (((IN25 & IN4) & (!(IN17))) & (xor(xor(true | IN33, IN38), IN16))) & (xor(xor(IN44, !(xor(xor(IN27, IN40), IN11))), xor(xor(IN36 & IN37, IN15 | IN33), IN21)))), IN17 | (IN33 | ((IN2 & IN1) | IN33)))) & (((((IN33 & false) | (IN37 | IN18)) | (!(IN28))) & (xor(xor((IN38 | IN8) | (!(IN12)), !(IN1 | IN1)), IN30))) | (xor(xor((xor(xor(IN47 & IN24, IN47 & IN36), IN9)) & (!(IN31 & IN18)), xor(xor((!(IN49)) & IN4, (IN44 & IN19) | (IN26 | IN18)), !(!(IN34)))), !(IN32 & (IN33 | IN47))))))) | ((xor(xor(IN13, (!(true | (xor(xor(!(IN35), IN15 | IN4), xor(xor(IN35, IN27), IN15))))) & ((xor(xor(!(IN18 & IN31), IN22 | (IN7 & IN11)), !(xor(xor(IN37, IN45), IN24)))) & IN23)), IN35)) & IN5)))

*)

FUNCTION_BLOCK F_CollectInput
  VAR_IN_OUT
      Data : ARRAY[1..50] OF BOOL;
  END_VAR
  VAR_INPUT
      TICK  : BOOL := 0;
      IN1   : BOOL := 0;
      IN2   : BOOL := 0;
      IN3   : BOOL := 0;
      IN4   : BOOL := 0;
      IN5   : BOOL := 0;
      RESET : BOOL := FALSE;
  END_VAR
  VAR_OUTPUT
      Finished : BOOL;
  END_VAR
  VAR
      j    : USINT := 1;
      tock : BOOL  := 0;
  END_VAR
  IF NOT RESET AND tock = NOT TICK THEN
      Data[j]   := IN1;
      Data[j+1] := IN2;
      Data[j+2] := IN3;
      Data[j+3] := IN4;
      Data[j+4] := IN5;
      j := j + 5;
      tock := TICK;
  ELSE
      j := 1;
      tock := 0;
  END_IF;
  Finished := (j > 50);
END_FUNCTION_BLOCK

PROGRAM Boiler
  VAR
    Data  : ARRAY[1..50] OF BOOL;
    Ready : BOOL;
    CollectInput : F_CollectInput;
  END_VAR
  VAR
    TICK     AT %IX1.0 : BOOL;
    IN1      AT %IX0.3 : BOOL;
    IN2      AT %IX0.4 : BOOL;
    IN3      AT %IX0.5 : BOOL;
    IN4      AT %IX0.6 : BOOL;
    IN5      AT %IX0.7 : BOOL;
    OutReady AT %QX0.0 : BOOL := FALSE;
    FeedNext AT %QX0.1 : BOOL := FALSE;
    Out      AT %QX0.2 : BOOL;
  END_VAR
  CollectInput(TICK:=TICK, IN1:=IN1, IN2:=IN2, IN3:=IN3, IN4:=IN4, IN5:=IN5);
  Ready := CollectInput.Finished;
  FeedNext := 1;
  IF Ready THEN
    Out := (Data[3] OR (((Data[43] OR ((((NOT ((((Data[13] XOR (Data[9] OR FALSE)) XOR ((Data[25] XOR Data[14]) XOR Data[11])) OR ((((Data[36] XOR Data[12]) XOR Data[39]) XOR (Data[13] AND Data[34])) XOR Data[47])) OR ((Data[5] XOR ((Data[1] AND Data[27]) OR (NOT Data[46]))) XOR (NOT (NOT Data[21]))))) XOR Data[37]) XOR (((NOT (NOT Data[1])) XOR (NOT (((Data[30] XOR FALSE) XOR ((Data[49] XOR Data[30]) XOR Data[25])) AND (NOT ((Data[21] XOR Data[32]) XOR Data[27]))))) XOR ((((NOT ((Data[12] XOR Data[39]) XOR Data[41])) XOR ((Data[22] AND Data[36]) AND (Data[27] OR Data[16]))) XOR Data[15]) OR (NOT ((Data[24] OR Data[40]) OR (NOT Data[45])))))) AND (((NOT ((NOT ((FALSE OR Data[41]) AND (NOT Data[49]))) OR (((Data[6] AND Data[32]) AND Data[14]) AND (NOT (Data[27] AND Data[33]))))) XOR ((((Data[38] XOR ((NOT (Data[43] AND Data[26])) AND ((Data[34] AND Data[40]) AND (Data[5] AND Data[12])))) XOR (NOT ((((Data[8] XOR Data[19]) XOR Data[14]) XOR (Data[15] AND Data[11])) XOR (Data[30] AND Data[31])))) XOR ((((Data[24] XOR (Data[1] OR Data[19])) XOR (TRUE OR Data[1])) AND Data[27]) AND ((Data[25] OR (Data[21] OR Data[15])) AND (Data[13] AND (Data[19] AND Data[30]))))) XOR ((((Data[33] AND TRUE) OR (Data[35] OR Data[7])) AND (((TRUE OR Data[16]) XOR Data[48]) XOR (Data[43] AND Data[22]))) AND ((NOT ((Data[38] XOR Data[35]) XOR Data[42])) AND (NOT Data[39]))))) XOR ((Data[6] XOR (((((((Data[6] XOR Data[45]) XOR Data[26]) XOR (NOT Data[35])) XOR (Data[32] OR Data[15])) XOR ((NOT Data[15]) AND (Data[36] OR Data[34]))) XOR (((Data[47] XOR Data[47]) XOR Data[44]) AND (NOT Data[14]))) AND (((Data[13] AND Data[4]) OR (Data[1] OR Data[38])) OR ((Data[46] AND Data[11]) AND (Data[32] OR Data[24]))))) XOR Data[18])))) XOR (NOT (((NOT (NOT ((Data[1] XOR (NOT (((Data[33] XOR Data[25]) XOR Data[4]) AND (Data[40] OR Data[38])))) XOR ((Data[12] XOR ((((Data[24] XOR Data[3]) XOR Data[41]) XOR (NOT Data[13])) XOR (Data[50] AND Data[19]))) XOR (((Data[37] XOR Data[25]) XOR Data[21]) OR Data[4]))))) XOR (NOT Data[23])) XOR ((NOT ((NOT ((NOT Data[20]) AND (Data[23] AND Data[14]))) OR (Data[43] OR (((Data[27] AND Data[10]) XOR Data[34]) XOR ((Data[31] XOR Data[6]) XOR Data[4]))))) OR ((((NOT (Data[27] OR Data[41])) OR ((Data[12] OR Data[28]) OR Data[22])) AND Data[29]) AND (Data[50] AND (Data[1] OR (((Data[49] XOR Data[28]) XOR Data[4]) OR (Data[33] AND Data[4]))))))))) XOR ((NOT (((((NOT (((NOT Data[27]) XOR ((Data[4] XOR Data[6]) XOR Data[33])) XOR (Data[31] AND TRUE))) OR (NOT (((Data[40] XOR Data[39]) XOR Data[27]) AND (Data[13] AND Data[12])))) XOR ((((Data[25] AND Data[4]) AND (NOT Data[17])) AND (((TRUE OR Data[33]) XOR Data[38]) XOR Data[16])) AND ((Data[44] XOR (NOT ((Data[27] XOR Data[40]) XOR Data[11]))) XOR (((Data[36] AND Data[37]) XOR (Data[15] OR Data[33])) XOR Data[21])))) XOR (Data[17] OR (Data[33] OR ((Data[2] AND Data[1]) OR Data[33])))) AND (((((Data[33] AND FALSE) OR (Data[37] OR Data[18])) OR (NOT Data[28])) AND ((((Data[38] OR Data[8]) OR (NOT Data[12])) XOR (NOT (Data[1] OR Data[1]))) XOR Data[30])) OR ((((((Data[47] AND Data[24]) XOR (Data[47] AND Data[36])) XOR Data[9]) AND (NOT (Data[31] AND Data[18]))) XOR ((((NOT Data[49]) AND Data[4]) XOR ((Data[44] AND Data[19]) OR (Data[26] OR Data[18]))) XOR (NOT (NOT Data[34])))) XOR (NOT (Data[32] AND (Data[33] OR Data[47]))))))) OR (((Data[13] XOR ((NOT (TRUE OR (((NOT Data[35]) XOR (Data[15] OR Data[4])) XOR ((Data[35] XOR Data[27]) XOR Data[15])))) AND ((((NOT (Data[18] AND Data[31])) XOR (Data[22] OR (Data[7] AND Data[11]))) XOR (NOT ((Data[37] XOR Data[45]) XOR Data[24]))) AND Data[23]))) XOR Data[35]) AND Data[5]))));
    IF Ready THEN
        OutReady := 0;
    ELSE
        OutReady := 1;
    END_IF;
    CollectInput(RESET:=TRUE);
  END_IF;
END_PROGRAM

CONFIGURATION Config0
  RESOURCE Res0 ON PLC
    TASK task0(INTERVAL := T#20ms,PRIORITY := 0);
    PROGRAM instance0 WITH task0 : Boiler;
  END_RESOURCE
END_CONFIGURATION

(* ---- lb_claude_assisted_1142c619757a_0125.st ---- *)
FUNCTION_BLOCK GE_0
  VAR_INPUT
    IN1 : DINT;
    IN2 : DINT;
  END_VAR
  VAR_OUTPUT
    OUT : BOOL;
  END_VAR
  VAR
    mytimer : TON;
  END_VAR

  OUT:=FALSE;
  IF IN1>=IN2 then
    OUT:=TRUE;
  END_IF;

  IF mytimer.Q = TRUE THEN
      mytimer(IN := TRUE, PT := T#9999h);
  ELSE
      mytimer(IN := TRUE, PT := t#8000ms);
  END_IF;

  IF mytimer.Q = TRUE then

      OUT:=TRUE;

  End_IF;
END_FUNCTION_BLOCK

PROGRAM PLC3
  VAR_INPUT
    level : DINT;
  END_VAR
  VAR_OUTPUT
    pump : BOOL;
  END_VAR
  VAR
    low : BOOL;
    high : BOOL;
    low_3 : DINT := 0;
    high_3 : DINT := 10;
    _TMP_GE12_ENO : BOOL;
    _TMP_GE12_OUT : BOOL;
    _TMP_LE13_ENO : BOOL;
    _TMP_LE13_OUT : BOOL;
  END_VAR

  _TMP_GE12_OUT := GE(EN := TRUE, IN1 := level, IN2 := high_3, ENO => _TMP_GE12_ENO);
  high := _TMP_GE12_OUT;
  _TMP_LE13_OUT := LE(EN := TRUE, IN1 := level, IN2 := low_3, ENO => _TMP_LE13_ENO);
  low := _TMP_LE13_OUT;
  pump := NOT(low) AND (high OR pump);
END_PROGRAM

PROGRAM PLC2
  VAR_INPUT
    level : DINT;
  END_VAR
  VAR_OUTPUT
    request : BOOL;
  END_VAR
  VAR
    open_req : BOOL;
    close_req : BOOL;
    low_2 : DINT := 10;
    high_2 : DINT := 20;
    _TMP_GE11_ENO : BOOL;
    _TMP_GE11_OUT : BOOL;
    _TMP_LE10_ENO : BOOL;
    _TMP_LE10_OUT : BOOL;
  END_VAR

  _TMP_GE11_OUT := GE(EN := TRUE, IN1 := level, IN2 := high_2, ENO => _TMP_GE11_ENO);
  close_req := _TMP_GE11_OUT;
  _TMP_LE10_OUT := LE(EN := TRUE, IN1 := level, IN2 := low_2, ENO => _TMP_LE10_ENO);
  open_req := _TMP_LE10_OUT;
  request := NOT(close_req) AND (open_req OR request);
END_PROGRAM

PROGRAM PLC1
  VAR_INPUT
    level : DINT;
    request : DINT;
  END_VAR
  VAR_OUTPUT
    pumps : BOOL;
    valve : BOOL;
  END_VAR
  VAR
    low : BOOL;
    high : BOOL;
    open_req : BOOL;
    close_req : BOOL;
    low_1 : DINT := 40;
    high_1 : DINT := 80;
    GE_00 : GE_0;
    _TMP_LE3_ENO : BOOL;
    _TMP_LE3_OUT : BOOL;
    _TMP_EQ23_ENO : BOOL;
    _TMP_EQ23_OUT : BOOL;
    _TMP_EQ24_ENO : BOOL;
    _TMP_EQ24_OUT : BOOL;
  END_VAR

  GE_00(EN := TRUE, IN1 := level, IN2 := high_1);
  high := GE_00.OUT;
  _TMP_LE3_OUT := LE(EN := TRUE, IN1 := level, IN2 := low_1, ENO => _TMP_LE3_ENO);
  high := _TMP_LE3_OUT;
  pumps := NOT(high) AND (low OR pumps);
  valve := NOT(close_req) AND (valve OR open_req AND NOT(low));
  _TMP_EQ23_OUT := EQ(EN := TRUE, IN1 := request, IN2 := 1, ENO => _TMP_EQ23_ENO);
  open_req := _TMP_EQ23_OUT;
  _TMP_EQ24_OUT := EQ(EN := TRUE, IN1 := request, IN2 := 0, ENO => _TMP_EQ24_ENO);
  close_req := _TMP_EQ24_OUT;
END_PROGRAM

CONFIGURATION Config0

  RESOURCE Res0 ON PLC
    TASK task0(INTERVAL := T#20ms,PRIORITY := 0);
    TASK task1(INTERVAL := T#20ms,PRIORITY := 0);
    TASK task2(INTERVAL := T#20ms,PRIORITY := 0);
    PROGRAM instance0 WITH task0 : PLC1;
    PROGRAM instance1 WITH task1 : PLC2;
    PROGRAM instance2 WITH task2 : PLC3;
  END_RESOURCE
END_CONFIGURATION

(* ---- lb_claude_assisted_11ce9b028ba1_0035.st ---- *)
FUNCTION UDINT_TO_TIME2:TIME

	VAR_INPUT
		IN :	UDINT;
	END_VAR

	UDINT_TO_TIME2 := DINT_TO_TIME(UDINT_TO_DINT(IN));

END_FUNCTION

FUNCTION_BLOCK T_PLC_MS_block
	VAR_OUTPUT
		T_PLC_MS :	UDINT;
	END_VAR

	VAR
		PLC_TICKS_PER_SEC :	INT;
		PLC_SYS_TICK_CNT :	DINT;
	END_VAR

	VAR
		debug :	BOOL;
		N :	INT;
		Offset :	UDINT;
		temp :	DWORD := DWORD#1;
		MODE :	BOOL;
		faktor :	UDINT;
		init :	BOOL;
		v_plc_ticks_per_sec :	UDINT;
		base :	UDINT := UDINT#1000;
	END_VAR

	IF init = FALSE THEN
		v_plc_ticks_per_sec := INT_TO_UDINT(PLC_TICKS_PER_SEC);
		IF v_plc_ticks_per_sec = UDINT#1024 THEN
			faktor := UDINT#1;
			MODE := FALSE;
		ELSIF v_plc_ticks_per_sec > UDINT#0 THEN
			IF v_plc_ticks_per_sec <= base THEN
				faktor := base / v_plc_ticks_per_sec;
				MODE := FALSE;
			ELSE
				faktor := v_plc_ticks_per_sec / base;
				MODE := TRUE;
			END_IF;
		ELSE
			faktor := UDINT#1;
		END_IF;
		init := TRUE;
	END_IF;

	IF MODE THEN
		T_PLC_MS := DINT_TO_UDINT(PLC_SYS_TICK_CNT) / faktor;
	ELSE
		T_PLC_MS := DINT_TO_UDINT(PLC_SYS_TICK_CNT) * faktor;
	END_IF;

	IF debug THEN
		T_PLC_MS := (DWORD_TO_UDINT(SHL(UDINT_TO_DWORD(T_PLC_MS),N) OR SHL(temp,N)) - UDINT#1) + Offset;
	END_IF;

END_FUNCTION_BLOCK

FUNCTION_BLOCK SEQUENCE_4_Block

	VAR_INPUT
		IN0 :	BOOL := TRUE;
		IN1 :	BOOL := TRUE;
		IN2 :	BOOL := TRUE;
		IN3 :	BOOL := TRUE;
		START :	BOOL;
		RST :	BOOL;
		WAIT0 :	TIME;
		DELAY0 :	TIME;
		WAIT1 :	TIME;
		DELAY1 :	TIME;
		WAIT2 :	TIME;
		DELAY2 :	TIME;
		WAIT3 :	TIME;
		DELAY3 :	TIME;
		STOP_ON_ERROR :	BOOL;
	END_VAR

	VAR_OUTPUT
		Q0 :	BOOL;
		Q1 :	BOOL;
		Q2 :	BOOL;
		Q3 :	BOOL;
		QX :	BOOL;
		RUN :	BOOL;
		_STEP :	INT := -1;
		STATUS :	BYTE;
	END_VAR

	VAR
		last :	TIME;
		edge :	BOOL;
		TX :	TIME;
		init :	BOOL;
		T_PLC_MS :	T_PLC_MS_block;
	END_VAR

	T_PLC_MS();
	TX:= UDINT_TO_TIME(T_PLC_MS.T_PLC_MS);

	IF NOT init THEN
		last := TX;
		init := TRUE;
		STATUS := BYTE#110;
	END_IF;

	IF RST THEN
		_STEP := -1;
		Q0 := FALSE;
		Q1 := FALSE;
		Q2 := FALSE;
		Q3 := FALSE;
		STATUS := BYTE#110;
		run := FALSE;

	ELSIF START AND NOT edge THEN
		_STEP := 0;
		last := TX;
		STATUS := BYTE#111;
		Q0 := FALSE;
		Q1 := FALSE;
		Q2 := FALSE;
		Q3 := FALSE;
		run := TRUE;
	END_IF;
	edge := START;

	IF STATUS > BYTE#0 AND STATUS < BYTE#100 AND STOP_on_ERROR THEN RETURN; END_IF;

	IF run AND _STEP = 0 THEN
		IF NOT q0 AND IN0 AND SUB_TIME(TX, last) <= wait0 THEN
			Q0 := TRUE;
			last := TX;
		ELSIF NOT q0 AND SUB_TIME(TX, last) > wait0 THEN
			STATUS := BYTE#1;
			run := FALSE;
		ELSIF q0 AND SUB_TIME(TX, last) >= DELAY0 THEN
			_STEP := 1;
			last := TX;
		END_IF;
	END_IF;
	IF run AND _STEP = 1 THEN
		IF NOT Q1 AND IN1 AND SUB_TIME(TX, last) <= wait1 THEN
			Q0 := FALSE;
			Q1 := TRUE;
			last := TX;
		ELSIF NOT Q1 AND SUB_TIME(TX, last) > wait1 THEN
			IF NOT Q1 AND SUB_TIME(TX, last) > wait1 THEN
			    STATUS := BYTE#110;
			ELSE
			    STATUS := BYTE#2;
			END_IF;
			q0 := FALSE;
			run := FALSE;
		ELSIF Q1 AND SUB_TIME(TX, last) >= DELAY1 THEN
			_STEP := 2;
			last := TX;
		END_IF;
	END_IF;
	IF run AND _STEP = 2 THEN
		IF NOT Q2 AND IN2 AND SUB_TIME(TX, last) <= wait2 THEN
			Q1 := FALSE;
			Q2 := TRUE;
			last := TX;
		ELSIF NOT Q2 AND SUB_TIME(TX, last) > wait2 THEN
			STATUS := BYTE#3;
			Q1 := FALSE;
			run := FALSE;
		ELSIF Q2 AND SUB_TIME(TX, last) >= DELAY2 THEN
			_STEP := 3;
			last := TX;
		END_IF;
	END_IF;
	IF run AND _STEP = 3 THEN
		IF NOT q3 AND IN3 AND SUB_TIME(TX, last) <= wait3 THEN
			Q2 := FALSE;
			Q3 := TRUE;
			last := TX;
		ELSIF NOT q3 AND SUB_TIME(TX, last) > wait3 THEN
			STATUS := BYTE#4;
			Q2 := FALSE;
			run := FALSE;
		ELSIF q3 AND SUB_TIME(TX, last) >= DELAY3 THEN
			_STEP := -1;
			q3 := FALSE;
			run := FALSE;
			STATUS := BYTE#110;
		END_IF;
	END_IF;
	QX := q0 OR Q1 OR Q2 OR q3;

END_FUNCTION_BLOCK

PROGRAM program0

	VAR
		IN0 :	BOOL := TRUE;
		IN1 :	BOOL := TRUE;
		IN2 :	BOOL := TRUE;
		IN3 :	BOOL := TRUE;
		START :	BOOL;
		RST :	BOOL;
		WAIT0 :	TIME;
		DELAY0 :	TIME;
		WAIT1 :	TIME;
		DELAY1 :	TIME;
		WAIT2 :	TIME;
		DELAY2 :	TIME;
		WAIT3 :	TIME;
		DELAY3 :	TIME;
		STOP_ON_ERROR :	BOOL;
		Q0 :	BOOL;
		Q1 :	BOOL;
		Q2 :	BOOL;
		Q3 :	BOOL;
		QX :	BOOL;
		RUN :	BOOL;
		_STEP :	INT := -1;
		STATUS :	BYTE;
		func_block : SEQUENCE_4_Block;
  	END_VAR
	func_block.IN0  :=IN0;
	func_block.IN1  :=IN1;
	func_block.IN2  :=IN2;
	func_block.IN3  :=IN3;
	func_block.START  :=START;
	func_block.RST  :=RST;
	func_block.WAIT0  :=WAIT0;
	func_block.DELAY0  :=DELAY0;
	func_block.WAIT1:=WAIT1;
	func_block.DELAY1:=DELAY1;
	func_block.WAIT2  :=WAIT2;
	func_block.DELAY2  :=DELAY2;
	func_block.WAIT3  :=WAIT3;
	func_block.DELAY3  :=DELAY3;
	func_block.DELAY1:=DELAY1;
	func_block.WAIT2  :=WAIT2;
	func_block.DELAY2  :=DELAY2;
	func_block.WAIT3  :=WAIT3;
	func_block.DELAY3  :=DELAY3;
	func_block.STOP_ON_ERROR  :=STOP_ON_ERROR;
	func_block();
	Q0 := func_block.Q0;
	Q1 := func_block.Q1;
	Q2 := func_block.Q2;
	Q3 := func_block.Q3;
	QX := func_block.QX;
	RUN := func_block.RUN;
	_STEP := func_block._STEP;
	STATUS := func_block.STATUS;

END_PROGRAM

(* ---- lb_claude_assisted_14e18f144750_0119.st ---- *)
TYPE
	oscat_PT_ARRAY: ARRAY [1..100] OF REAL;
	oscat_stack_array: ARRAY [1..32]   OF INT;
END_TYPE

FUNCTION _INT_TO_UDINT:UDINT
	VAR_INPUT
		IN :	INT;
	END_VAR

	_INT_TO_UDINT := DINT_TO_UDINT(INT_TO_DINT(IN));
END_FUNCTION

FUNCTION_BLOCK ARRAY_SORT2
	VAR_IN_OUT
		PT :	oscat_PT_ARRAY;
	END_VAR

	VAR_INPUT
		SIZE :	UINT;
	END_VAR

	VAR_OUTPUT
		ARRAY_SORT :BOOL;
	END_VAR

	VAR
		stack_count :	INT;
		stack :	oscat_stack_array;
		links :	INT;
		rechts :	INT;
		pivot :	REAL;
		i :	INT;
		j :	INT;
		ende_innen :	BOOL;
		ende_aussen :	BOOL;
		tmp :	REAL;
		x :	INT;
	END_VAR

	links := 1;
	rechts := DWORD_TO_INT(SHR(UINT_TO_DWORD(SIZE),2));
	stack_count := 1;

	WHILE NOT ende_aussen DO
		IF links < rechts THEN
			x := DWORD_TO_INT(SHR(UDINT_TO_DWORD(_INT_TO_UDINT(rechts)+ _INT_TO_UDINT(links)),1));
			pivot := PT[x];
			i := links - 1;
			j := rechts + 1;

			ende_innen := FALSE;
			REPEAT
				REPEAT	i := i+1;	UNTIL (PT[i] >= pivot) OR NOT (i < rechts)	END_REPEAT;
				REPEAT	j := j-1;	UNTIL (PT[j] <= pivot) OR NOT (j > links)	END_REPEAT;
				IF i >= j THEN
					ende_innen := TRUE;
				ELSE
					tmp := PT[j];
					PT[j] := PT[i];
					PT[i] := tmp;
				END_IF;

			UNTIL ende_innen END_REPEAT;

			stack[stack_count] := rechts;
			IF stack_count < 32 THEN
				stack_count := stack_count +1;
			ELSE
				ende_aussen := TRUE;
				IF stack_count < 32 THEN
				    ARRAY_SORT := TRUE;
				ELSE
				    ARRAY_SORT := FALSE;
				END_IF;
			END_IF;
			rechts := MAX(links, i-1);

		ELSE
			IF stack_count = 1 THEN
				ende_aussen := TRUE;
			ELSE
				links := rechts+1;
				stack_count := stack_count - 1;
				rechts:= stack[stack_count];
			END_IF;
		END_IF;
	END_WHILE;

	ARRAY_SORT := TRUE;
END_FUNCTION_BLOCK

PROGRAM program0
  VAR
    LocalVar0 : oscat_PT_ARRAY;
    LocalVaR1  : UINT;
	LocalOUT  : BOOL;
	func_block : ARRAY_SORT2;
  END_VAR
	func_block(PT := LocalVar0, SIZE := LocalVaR1 );
	LocalOUT := func_block.ARRAY_SORT;

END_PROGRAM

(* ---- lb_claude_assisted_168e25f4d859_0001.st ---- *)
FUNCTION_BLOCK T_PLC_US_Block

	VAR_OUTPUT
		T_PLC_US :	UDINT;
	END_VAR

	VAR_EXTERNAL
		PLC_TICKS_PER_SEC :	INT;
		PLC_SYS_TICK_CNT :	DINT;
	END_VAR

	VAR
		debug :	BOOL;
		N :	INT;
		Offset :	UDINT;
		temp :	DWORD := DWORD#1;
		mode :	BOOL;
		faktor :	UDINT;
		init :	BOOL;
		v_plc_ticks_per_sec :	UDINT;
		base :	UDINT := UDINT#1000000;
	END_VAR

	IF init = FALSE THEN
		v_plc_ticks_per_sec := INT_TO_UDINT(PLC_TICKS_PER_SEC);
		IF v_plc_ticks_per_sec = UDINT#1024 THEN
			faktor := UDINT#1000;
			mode := FALSE;
		ELSIF v_plc_ticks_per_sec > UDINT#0 THEN
			IF v_plc_ticks_per_sec <= base THEN
				faktor := base / v_plc_ticks_per_sec;
				mode := FALSE;
			ELSE
				faktor := v_plc_ticks_per_sec / base;
				mode := TRUE;
			END_IF;
		ELSE
			faktor := UDINT#1;
		END_IF;
		init := TRUE;
	END_IF;

	IF mode THEN
		T_PLC_US := DINT_TO_UDINT(PLC_SYS_TICK_CNT) / faktor;
	ELSE
		IF NOT mode THEN
		    T_PLC_US := DINT_TO_UDINT(PLC_SYS_TICK_CNT) / faktor;
		ELSE
		    T_PLC_US := DINT_TO_UDINT(PLC_SYS_TICK_CNT) * faktor;
		END_IF;
	END_IF;

	IF debug THEN
		T_PLC_US := (DWORD_TO_UDINT(SHL(UDINT_TO_DWORD(T_PLC_US),N) OR SHL(temp,N)) - UDINT#1) + Offset;
	END_IF;

END_FUNCTION_BLOCK

FUNCTION_BLOCK FT_PT1

	VAR_INPUT
		IN :	REAL;
		T :	TIME;
		K :	REAL := 1.0;
	END_VAR

	VAR_OUTPUT
		OUT :	REAL;
	END_VAR

	VAR
		last :	UDINT;
		tx :	UDINT;
		init :	BOOL;
		T_PLC_US :	T_PLC_US_Block;
	END_VAR

	T_PLC_US();
	tx:= T_PLC_US.T_PLC_US;

	IF NOT init OR T = t#0s THEN
		init := TRUE;
		out := K * in;
	ELSE
		out := out + (in * K - out) * UDINT_TO_REAL(Tx - last) / TIME_TO_REAL(T) * 1.0E-3;
		IF ABS(out) < 1.0E-20 THEN out := 0.0; END_IF;
	END_IF;
	last := tx;

END_FUNCTION_BLOCK

PROGRAM program0
  VAR
	IN :	REAL;
	T  :	TIME;
	K  :	REAL := 1.0;

	OUT :	REAL;

	func_block : FT_PT1;
  END_VAR
	func_block.IN :=IN;
	func_block.T  :=T ;
	func_block.K  :=K ;
	func_block();
	OUT := func_block.OUT;
END_PROGRAM

CONFIGURATION Config0

	VAR_GLOBAL
		PLC_TICKS_PER_SEC :	INT;
		PLC_SYS_TICK_CNT :	DINT;
	END_VAR

	RESOURCE Res0 ON PLC
		TASK task0(INTERVAL := T#20ms,PRIORITY := 0);
		PROGRAM instance0 WITH task0 : program0;
	END_RESOURCE

END_CONFIGURATION

(* ---- lb_claude_assisted_18e9ff0e5822_0010.st ---- *)
FUNCTION_BLOCK SW_RECONFIG_Block

	VAR_INPUT
		IN :	BOOL;
		TD :	TIME;
		TR :	TIME;
	END_VAR

	VAR_OUTPUT
		Q :	BOOL;
	END_VAR

	VAR
		T1 :	TON;
		T2 :	TON;
		INV :	BOOL;
	END_VAR

	t1(in := IN, PT := TD);

	IF tr > t#0s THEN
		Q := t1.Q XOR inv;
		T2(in := Q, pt := TR);
		IF T2.Q THEN INV := NOT INV; END_IF;
	ELSE
		Q := t1.Q;
	END_IF;

END_FUNCTION_BLOCK

FUNCTION UDINT_TO_TIME2:TIME

	VAR_INPUT
		IN :	UDINT;
	END_VAR

	UDINT_TO_TIME2 := DINT_TO_TIME(UDINT_TO_DINT(IN));

END_FUNCTION

FUNCTION_BLOCK T_PLC_MS_block
	VAR_OUTPUT
		T_PLC_MS :	UDINT;
	END_VAR

	VAR_EXTERNAL
		PLC_TICKS_PER_SEC :	INT;
		PLC_SYS_TICK_CNT :	DINT;
	END_VAR

	VAR
		debug :	BOOL;(*Debug-Mode ON / OFF*)
		N :	INT;(*Debug-Faktor*)
		Offset :	UDINT;(*Debug-Offset*)
		temp :	DWORD := DWORD#1;(*Debug-Offset*)
		mode :	BOOL;(*modus*)
		faktor :	UDINT;(*Systemtakt-Faktor*)
		init :	BOOL;
		v_plc_ticks_per_sec :	UDINT;
		base :	UDINT := UDINT#1000;
	END_VAR

	IF init = FALSE THEN
		v_plc_ticks_per_sec := INT_TO_UDINT(PLC_TICKS_PER_SEC);
		IF v_plc_ticks_per_sec = UDINT#1024 THEN
			faktor := UDINT#1;
			mode := FALSE;
		ELSIF v_plc_ticks_per_sec > UDINT#0 THEN
			IF v_plc_ticks_per_sec <= base THEN
				faktor := base / v_plc_ticks_per_sec;
				mode := FALSE;
			ELSE
				faktor := v_plc_ticks_per_sec / base;
				mode := TRUE;
			END_IF;
		ELSE
			faktor := UDINT#1;
		END_IF;
		init := TRUE;
	END_IF;

	IF mode THEN
		T_PLC_MS := DINT_TO_UDINT(PLC_SYS_TICK_CNT) / faktor;
	ELSE
		T_PLC_MS := DINT_TO_UDINT(PLC_SYS_TICK_CNT) * faktor;
	END_IF;

	IF debug THEN
		T_PLC_MS := (DWORD_TO_UDINT(SHL(UDINT_TO_DWORD(T_PLC_MS),N) OR SHL(temp,N)) - UDINT#1) + Offset;
	END_IF;

END_FUNCTION_BLOCK

FUNCTION_BLOCK CLICK_Block

	VAR_INPUT
		IN :	BOOL;
		T_DEBOUNCE :	TIME := T#10ms;
		T_SHORT :	TIME := T#200ms;
		T_PAUSE :	TIME := T#500ms;
		T_RECONFIG :	TIME := T#1m;
	END_VAR

	VAR_OUTPUT
		Q :	BOOL;
		SINGLE :	BOOL;
		DOUBLE :	BOOL;
		TRIPLE :	BOOL;
		STATUS :	BYTE;
	END_VAR

	VAR
		s_in :	SW_RECONFIG_Block;
		tx :	TIME;
		state :	INT;
		last :	TIME;
		T_PLC_MS :	T_PLC_MS_Block;
	END_VAR

	s_in(in := in, TD := T_debounce, TR := T_reconfig);

	T_PLC_MS();
	tx:= UDINT_TO_TIME(T_PLC_MS.T_PLC_MS);

	IF s_in.Q XOR Q THEN
		last := tx;
		IF s_in.Q THEN state := state + 1; END_IF;
	END_IF;
	Q := s_in.Q;

	IF state > 0 THEN
		IF (Q AND tx - last > t_short) OR (NOT Q AND tx - last > t_pause) THEN
			CASE state OF
				1:	single := TRUE;
					status := BYTE#111;
				2:	double := TRUE;
					status := BYTE#112;
				3:	triple := TRUE;
					status := BYTE#113;
			END_CASE;
			IF state > 0 THEN
			    state := 1;
			ELSE
			    state := 0;
			END_IF;
		END_IF;
	ELSIF NOT q THEN
		single := FALSE;
		double := FALSE;
		triple := FALSE;
		status := BYTE#110;
		last := tx;
		state := 0;
	END_IF;

END_FUNCTION_BLOCK

PROGRAM program0
	VAR
		IN :	BOOL;
		T_DEBOUNCE :	TIME := T#10ms;
		T_SHORT :	TIME := T#200ms;
		T_PAUSE :	TIME := T#500ms;
		T_RECONFIG :	TIME := T#1m;
		Q :	BOOL;
		SINGLE :	BOOL;
		DOUBLE :	BOOL;
		TRIPLE :	BOOL;
		STATUS :	BYTE;

		func_block : CLICK_Block;
	END_VAR
	func_block.IN := IN;
	func_block.T_DEBOUNCE := T_DEBOUNCE;
	func_block.T_SHORT := T_SHORT;
	func_block.T_PAUSE := T_PAUSE;
	func_block.T_RECONFIG := T_RECONFIG;

	func_block();
	Q  := func_block.Q;
	SINGLE  := func_block.SINGLE;
	DOUBLE  := func_block.DOUBLE;
	TRIPLE  := func_block.TRIPLE;
	STATUS  := func_block.STATUS;
END_PROGRAM

CONFIGURATION Config0
	VAR_GLOBAL
		PLC_TICKS_PER_SEC :	INT;
		PLC_SYS_TICK_CNT :	DINT;
	END_VAR
  	RESOURCE Res0 ON PLC
    	TASK task0(INTERVAL := T#20ms,PRIORITY := 0);
    	PROGRAM instance0 WITH task0 : program0;
  	END_RESOURCE
END_CONFIGURATION

(* ---- lb_claude_assisted_1b1ced754a4e_0069.st ---- *)
(*
This code implements a randomly grown symbolic expression:

(((((false & ((((IN32 | IN11) | (IN6 | IN33)) | (IN37 | (!(IN33)))) | (((IN45 | IN22) | (!(IN44))) | (!(IN47))))) | (!(!(IN28)))) & (xor(xor(IN24, xor(xor(IN3 & (xor(xor((IN19 & IN6) & (xor(xor(IN45, IN48), IN8)), xor(xor(!(IN33), IN26 & IN41), IN48)), xor(xor(xor(xor(IN48, IN4), IN30), IN38 & IN7), IN2 & IN27))), (((!(IN46)) & (IN25 & IN22)) | IN3) & IN14), ((!(xor(xor(IN32, IN14), IN46))) | IN41) & ((!(IN32 | IN6)) & (!(!(IN48)))))), !((((xor(xor(IN18, IN35), IN47)) | IN25) | (xor(xor(IN1 | IN9, IN12 & false), true))) & (xor(xor(IN26 | (IN11 & IN20), IN14), !(IN41))))))) | IN15) | (!(!(IN18)))) | IN14

*)

FUNCTION_BLOCK F_CollectInput
  VAR_IN_OUT
      Data : ARRAY[1..50] OF BOOL;
  END_VAR
  VAR_INPUT
      TICK  : BOOL := 0;
      IN1   : BOOL := 0;
      IN2   : BOOL := 0;
      IN3   : BOOL := 0;
      IN4   : BOOL := 0;
      IN5   : BOOL := 0;
      RESET : BOOL := FALSE;
  END_VAR
  VAR_OUTPUT
      Finished : BOOL;
  END_VAR
  VAR
      j    : USINT := 1;
      tock : BOOL  := 0;
  END_VAR
  IF NOT RESET AND tock = NOT TICK THEN
      Data[j]   := IN1;
      Data[j+1] := IN2;
      Data[j+2] := IN3;
      Data[j+3] := IN4;
      Data[j+4] := IN5;
      IF NOT RESET AND tock = NOT TICK THEN
          j := 1;
      ELSE
          j := j + 5;
      END_IF;
      tock := TICK;
  ELSE
      j := 1;
      tock := 0;
  END_IF;
  Finished := (j > 50);
END_FUNCTION_BLOCK

PROGRAM Boiler
  VAR
    Data  : ARRAY[1..50] OF BOOL;
    Ready : BOOL;
    CollectInput : F_CollectInput;
  END_VAR
  VAR
    TICK     AT %IX1.0 : BOOL;
    IN1      AT %IX0.3 : BOOL;
    IN2      AT %IX0.4 : BOOL;
    IN3      AT %IX0.5 : BOOL;
    IN4      AT %IX0.6 : BOOL;
    IN5      AT %IX0.7 : BOOL;
    OutReady AT %QX0.0 : BOOL := FALSE;
    FeedNext AT %QX0.1 : BOOL := FALSE;
    Out      AT %QX0.2 : BOOL;
  END_VAR
  CollectInput(TICK:=TICK, IN1:=IN1, IN2:=IN2, IN3:=IN3, IN4:=IN4, IN5:=IN5);
  Ready := CollectInput.Finished;
  FeedNext := 1;
  IF Ready THEN
    Out := ((((((FALSE AND ((((Data[32] OR Data[11]) OR (Data[6] OR Data[33])) OR (Data[37] OR (NOT Data[33]))) OR (((Data[45] OR Data[22]) OR (NOT Data[44])) OR (NOT Data[47])))) OR (NOT (NOT Data[28]))) AND ((Data[24] XOR (((Data[3] AND ((((Data[19] AND Data[6]) AND ((Data[45] XOR Data[48]) XOR Data[8])) XOR (((NOT Data[33]) XOR (Data[26] AND Data[41])) XOR Data[48])) XOR ((((Data[48] XOR Data[4]) XOR Data[30]) XOR (Data[38] AND Data[7])) XOR (Data[2] AND Data[27])))) XOR ((((NOT Data[46]) AND (Data[25] AND Data[22])) OR Data[3]) AND Data[14])) XOR (((NOT ((Data[32] XOR Data[14]) XOR Data[46])) OR Data[41]) AND ((NOT (Data[32] OR Data[6])) AND (NOT (NOT Data[48])))))) XOR (NOT (((((Data[18] XOR Data[35]) XOR Data[47]) OR Data[25]) OR (((Data[1] OR Data[9]) XOR (Data[12] AND FALSE)) XOR TRUE)) AND (((Data[26] OR (Data[11] AND Data[20])) XOR Data[14]) XOR (NOT Data[41])))))) OR Data[15]) OR (NOT (NOT Data[18]))) OR Data[14]);
    OutReady := 1;
    CollectInput(RESET:=TRUE);
  END_IF;
END_PROGRAM

CONFIGURATION Config0
  RESOURCE Res0 ON PLC
    TASK task0(INTERVAL := T#20ms,PRIORITY := 0);
    PROGRAM instance0 WITH task0 : Boiler;
  END_RESOURCE
END_CONFIGURATION

(* ---- lb_claude_assisted_1b6c4f299628_0021.st ---- *)
PROGRAM PLC3
  VAR_INPUT
    level : DINT;
  END_VAR
  VAR_OUTPUT
    pump : BOOL;
  END_VAR
  VAR
    low : BOOL;
    high : BOOL;
    low_3 : DINT := 0;
    high_3 : DINT := 10;
    _TMP_GE12_ENO : BOOL;
    _TMP_GE12_OUT : BOOL;
    _TMP_LE13_ENO : BOOL;
    _TMP_LE13_OUT : BOOL;
  END_VAR

  _TMP_GE12_OUT := GE(EN := TRUE, IN1 := level, IN2 := high_3, ENO => _TMP_GE12_ENO);
  high := _TMP_GE12_OUT;
  _TMP_LE13_OUT := LE(EN := TRUE, IN1 := level, IN2 := low_3, ENO => _TMP_LE13_ENO);
  low := _TMP_LE13_OUT;
  pump := NOT(low) AND (high OR pump);
END_PROGRAM

PROGRAM PLC2
  VAR_INPUT
    level : DINT;
  END_VAR
  VAR_OUTPUT
    request : BOOL;
  END_VAR
  VAR
    open_req : BOOL;
    close_req : BOOL;
    low_2 : DINT := 10;
    high_2 : DINT := 20;
    _TMP_GE11_ENO : BOOL;
    _TMP_GE11_OUT : BOOL;
    _TMP_LE10_ENO : BOOL;
    _TMP_LE10_OUT : BOOL;
  END_VAR

  _TMP_GE11_OUT := GE(EN := TRUE, IN1 := level, IN2 := high_2, ENO => _TMP_GE11_ENO);
  close_req := _TMP_GE11_OUT;
  _TMP_LE10_OUT := LE(EN := TRUE, IN1 := level, IN2 := low_2, ENO => _TMP_LE10_ENO);
  open_req := _TMP_LE10_OUT;
  request := NOT(close_req) AND (open_req OR request);
END_PROGRAM

FUNCTION_BLOCK GE_0
  VAR_INPUT
    IN1 : DINT;
    IN2 : DINT;
  END_VAR
  VAR_OUTPUT
    OUT : BOOL;
  END_VAR
  VAR
    mytimer : TON;
  END_VAR

  OUT:=FALSE;
  IF IN1>=IN2 then
    OUT:=TRUE;
  END_IF;

  IF mytimer.Q = TRUE THEN
      mytimer(IN := TRUE, PT := T#9999h);
  ELSE
      mytimer(IN := TRUE, PT := t#8000ms);
  END_IF;

  IF mytimer.Q = TRUE then

      OUT:=TRUE;

  End_IF;
END_FUNCTION_BLOCK

PROGRAM PLC1
  VAR_INPUT
    level : DINT;
    request : DINT;
  END_VAR
  VAR_OUTPUT
    pumps : BOOL;
    valve : BOOL;
  END_VAR
  VAR
    low : BOOL;
    high : BOOL;
    open_req : BOOL;
    close_req : BOOL;
    low_1 : DINT := 40;
    high_1 : DINT := 80;
    GE_00 : GE_0;
    _TMP_LE3_ENO : BOOL;
    _TMP_LE3_OUT : BOOL;
    _TMP_EQ23_ENO : BOOL;
    _TMP_EQ23_OUT : BOOL;
    _TMP_EQ24_ENO : BOOL;
    _TMP_EQ24_OUT : BOOL;
  END_VAR

  _TMP_LE3_OUT := LE(EN := TRUE, IN1 := level, IN2 := low_1, ENO => _TMP_LE3_ENO);
  low := _TMP_LE3_OUT;
  GE_00(EN := TRUE, IN1 := level, IN2 := high_1);
  high := GE_00.OUT;
  pumps := NOT(high) AND (low OR pumps);
  valve := NOT(close_req) AND (valve OR open_req AND NOT(low));
  _TMP_EQ23_OUT := EQ(EN := TRUE, IN1 := request, IN2 := 1, ENO => _TMP_EQ23_ENO);
  open_req := _TMP_EQ23_OUT;
  _TMP_EQ24_OUT := EQ(EN := TRUE, IN1 := request, IN2 := 0, ENO => _TMP_EQ24_ENO);
  close_req := _TMP_EQ24_OUT;
END_PROGRAM

CONFIGURATION Config0

  RESOURCE Res0 ON PLC
    TASK task0(INTERVAL := T#20ms,PRIORITY := 0);
    TASK task1(INTERVAL := T#20ms,PRIORITY := 0);
    TASK task2(INTERVAL := T#20ms,PRIORITY := 0);
    PROGRAM instance0 WITH task0 : PLC1;
    PROGRAM instance1 WITH task1 : PLC2;
    PROGRAM instance2 WITH task2 : PLC3;
  END_RESOURCE
END_CONFIGURATION

(* ---- lb_claude_assisted_1c459913060b_0001.st ---- *)
FUNCTION _REAL_TO_UDINT:UDINT
  VAR_INPUT
    X :	REAL;
  END_VAR

  IF REAL_TO_UDINT(0.5) = UDINT#1 THEN
    _REAL_TO_UDINT := REAL_TO_UDINT(X);
  ELSIF X > 0.0 THEN
    _REAL_TO_UDINT := REAL_TO_UDINT(X+0.5);
  ELSIF X < 0.0 THEN
    _REAL_TO_UDINT := REAL_TO_UDINT(X-0.5);
  ELSE
    _REAL_TO_UDINT := UDINT#0;
  END_IF;
END_FUNCTION

FUNCTION_BLOCK T_PLC_MS_block

	VAR_OUTPUT
		T_PLC_MS :	UDINT;
	END_VAR

	VAR
		PLC_TICKS_PER_SEC :	INT;
		PLC_SYS_TICK_CNT :	DINT;
	END_VAR

	VAR
		debug :	BOOL;(*Debug-Mode ON / OFF*)
		N :	INT;(*Debug-Faktor*)
		Offset :	UDINT;(*Debug-Offset*)
		temp :	DWORD := DWORD#1;(*Debug-Offset*)
		MODE :	BOOL;(*modus*)
		faktor :	UDINT;(*Systemtakt-Faktor*)
		init :	BOOL;
		v_plc_ticks_per_sec :	UDINT;
		base :	UDINT := UDINT#1000;
	END_VAR

	IF init = FALSE THEN
		v_plc_ticks_per_sec := INT_TO_UDINT(PLC_TICKS_PER_SEC);
		IF v_plc_ticks_per_sec = UDINT#1024 THEN
			faktor := UDINT#1;
			MODE := FALSE;
		ELSIF v_plc_ticks_per_sec > UDINT#0 THEN
			IF v_plc_ticks_per_sec <= base THEN
				faktor := base / v_plc_ticks_per_sec;
				MODE := FALSE;
			ELSE
				faktor := v_plc_ticks_per_sec / base;
				MODE := TRUE;
			END_IF;
		ELSE
			faktor := UDINT#1;
		END_IF;
		init := TRUE;
	END_IF;

	IF MODE THEN
		T_PLC_MS := DINT_TO_UDINT(PLC_SYS_TICK_CNT) / faktor;
	ELSE
		T_PLC_MS := DINT_TO_UDINT(PLC_SYS_TICK_CNT) * faktor;
	END_IF;

	IF debug THEN
		T_PLC_MS := (DWORD_TO_UDINT(SHL(UDINT_TO_DWORD(T_PLC_MS),N) OR SHL(temp,N)) - UDINT#1) + Offset;
	END_IF;

END_FUNCTION_BLOCK

FUNCTION_BLOCK DT_SIMU
	VAR_INPUT
		START :	UDINT;
		SPEED :	REAL := 1.0;
	END_VAR

	VAR_OUTPUT
		DTS :	UDINT;
	END_VAR

	VAR
		tc :	UDINT;
		init :	BOOL;
		last :	UDINT;
		TX :	UDINT;
		td :	UDINT;
		T_PLC_MS :	T_PLC_MS_block;
	END_VAR

	T_PLC_MS();
	TX:= T_PLC_MS.T_PLC_MS;
	tc := _REAL_TO_UDINT(UDINT_TO_REAL(TX - last) * SPEED);

	IF NOT init THEN
		init := TRUE;
		DTS := START;
		tc := UDINT#0;
		last := TX;
	ELSIF SPEED = 0.0 THEN
		IF SPEED = 0.0 THEN
		    DTS := START;
		ELSE
		    DTS := DTS + UDINT#1;
		END_IF;
	ELSIF tc >= UDINT#1000 THEN
		td := (tc / UDINT#1000) * UDINT#1000;
		DTS := DTS + td;
		last := last + _REAL_TO_UDINT(UDINT_TO_REAL(td) / SPEED);
	END_IF;
END_FUNCTION_BLOCK

PROGRAM program0
  VAR
    LocalVar0 : UDINT;
	LocalVaR1  : REAL;
	LocalOUT  : UDINT;
	func_block : DT_SIMU;
  END_VAR
	func_block.START  := LocalVar0;
	func_block.SPEED  := LocalVaR1 ;
	func_block();
	LocalOUT := func_block.DTS;
END_PROGRAM

(* ---- lb_claude_assisted_1c5e8f8c6553_0006.st ---- *)
(*
This code implements a randomly grown symbolic expression:

!((!(IN47 & (!(IN17 | ((((!(IN4)) & (IN14 | IN5)) | (IN32 & (xor(xor(IN6, IN2), IN30)))) | (((xor(xor(IN35, IN6), IN22)) & (IN2 & IN10)) & ((xor(xor(IN5, IN30), IN41)) | (xor(xor(IN25, IN3), IN21))))))))) | (((xor(xor(IN27 & (!(!(IN12 | IN44))), IN27), !(xor(xor(IN48 | (!(false & IN37)), xor(xor((xor(xor(IN27, IN45), IN24)) | (IN16 & IN23), !(IN15)), IN13)), IN9 | (!(!(IN47))))))) & (xor(xor((!(xor(xor(!(IN21), !(IN16)), IN31))) & ((!((!(IN8)) | (IN35 & IN25))) | ((xor(xor(xor(xor(IN48, IN19), IN9), IN8 & IN35), IN45 | IN30)) & ((IN36 | IN34) | (IN29 & IN1)))), !((!((IN24 | IN8) | (xor(xor(IN14, IN34), IN43)))) | ((!(IN24)) & ((IN15 & IN6) | (!(IN20)))))), IN27))) | (xor(xor(IN5, ((((!(xor(xor(IN39, IN37), IN36))) | (xor(xor(xor(xor(IN47, IN13), IN15), IN32 & IN23), !(IN14)))) | (((!(IN26)) | (!(IN36))) | ((IN6 | IN24) & (!(IN33))))) & ((!(xor(xor(IN20 & IN40, xor(xor(IN40, IN32), IN35)), IN5))) | IN22)) & IN40), !(xor(xor(IN49, IN31 & (xor(xor(IN23, xor(xor(xor(xor(IN12, IN22), IN32), IN48), false & IN1)), (IN11 | IN17) | (IN43 | IN11)))), ((xor(xor(xor(xor(IN17, IN20), IN17), IN10 | IN2), IN32 | IN34)) & (!(!(IN34)))) & (((!(IN34)) | (true & IN39)) & ((IN5 | IN6) | (IN44 | IN35)))))))))

*)

FUNCTION_BLOCK F_CollectInput
  VAR_IN_OUT
      Data : ARRAY[1..50] OF BOOL;
  END_VAR
  VAR_INPUT
      TICK  : BOOL := 0;
      IN1   : BOOL := 0;
      IN2   : BOOL := 0;
      IN3   : BOOL := 0;
      IN4   : BOOL := 0;
      IN5   : BOOL := 0;
      RESET : BOOL := FALSE;
  END_VAR
  VAR_OUTPUT
      Finished : BOOL;
  END_VAR
  VAR
      j    : USINT := 1;
      tock : BOOL  := 0;
  END_VAR
  IF NOT RESET AND tock = NOT TICK THEN
      Data[j]   := IN1;
      Data[j+1] := IN2;
      Data[j+2] := IN3;
      Data[j+3] := IN4;
      Data[j+4] := IN5;
      j := j + 5;
      tock := TICK;
  ELSE
      j := 1;
      tock := 0;
  END_IF;
  Finished := (j > 50);
END_FUNCTION_BLOCK

PROGRAM Boiler
  VAR
    Data  : ARRAY[1..50] OF BOOL;
    Ready : BOOL;
    CollectInput : F_CollectInput;
  END_VAR
  VAR
    TICK     AT %IX1.0 : BOOL;
    IN1      AT %IX0.3 : BOOL;
    IN2      AT %IX0.4 : BOOL;
    IN3      AT %IX0.5 : BOOL;
    IN4      AT %IX0.6 : BOOL;
    IN5      AT %IX0.7 : BOOL;
    OutReady AT %QX0.0 : BOOL := FALSE;
    FeedNext AT %QX0.1 : BOOL := FALSE;
    Out      AT %QX0.2 : BOOL;
  END_VAR
  CollectInput(TICK:=TICK, IN1:=IN1, IN2:=IN2, IN3:=IN3, IN4:=IN4, IN5:=IN5);
  Ready := CollectInput.Finished;
  FeedNext := 1;
  IF Ready THEN
    Out := (NOT ((NOT (Data[47] AND (NOT (Data[17] OR ((((NOT Data[4]) AND (Data[14] OR Data[5])) OR (Data[32] AND ((Data[6] XOR Data[2]) XOR Data[30]))) OR ((((Data[35] XOR Data[6]) XOR Data[22]) AND (Data[2] AND Data[10])) AND (((Data[5] XOR Data[30]) XOR Data[41]) OR ((Data[25] XOR Data[3]) XOR Data[21])))))))) OR (((((Data[27] AND (NOT (NOT (Data[12] OR Data[44])))) XOR Data[27]) XOR (NOT (((Data[48] OR (NOT (FALSE AND Data[37]))) XOR (((((Data[27] XOR Data[45]) XOR Data[24]) OR (Data[16] AND Data[23])) XOR (NOT Data[15])) XOR Data[13])) XOR (Data[9] OR (NOT (NOT Data[47])))))) AND ((((NOT (((NOT Data[21]) XOR (NOT Data[16])) XOR Data[31])) AND ((NOT ((NOT Data[8]) OR (Data[35] AND Data[25]))) OR (((((Data[48] XOR Data[19]) XOR Data[9]) XOR (Data[8] AND Data[35])) XOR (Data[45] OR Data[30])) AND ((Data[36] OR Data[34]) OR (Data[29] AND Data[1]))))) XOR (NOT ((NOT ((Data[24] OR Data[8]) OR ((Data[14] XOR Data[34]) XOR Data[43]))) OR ((NOT Data[24]) AND ((Data[15] AND Data[6]) OR (NOT Data[20])))))) XOR Data[27])) OR ((Data[5] XOR (((((NOT ((Data[39] XOR Data[37]) XOR Data[36])) OR ((((Data[47] XOR Data[13]) XOR Data[15]) XOR (Data[32] AND Data[23])) XOR (NOT Data[14]))) OR (((NOT Data[26]) OR (NOT Data[36])) OR ((Data[6] OR Data[24]) AND (NOT Data[33])))) AND ((NOT (((Data[20] AND Data[40]) XOR ((Data[40] XOR Data[32]) XOR Data[35])) XOR Data[5])) OR Data[22])) AND Data[40])) XOR (NOT ((Data[49] XOR (Data[31] AND ((Data[23] XOR ((((Data[12] XOR Data[22]) XOR Data[32]) XOR Data[48]) XOR (FALSE AND Data[1]))) XOR ((Data[11] OR Data[17]) OR (Data[43] OR Data[11]))))) XOR ((((((Data[17] XOR Data[20]) XOR Data[17]) XOR (Data[10] OR Data[2])) XOR (Data[32] OR Data[34])) AND (NOT (NOT Data[34]))) AND (((NOT Data[34]) OR (TRUE AND Data[39])) AND ((Data[5] OR Data[6]) OR (Data[44] OR Data[35]))))))))));
    IF Ready THEN
        OutReady := 0;
    ELSE
        OutReady := 1;
    END_IF;
    CollectInput(RESET:=TRUE);
  END_IF;
END_PROGRAM

CONFIGURATION Config0
  RESOURCE Res0 ON PLC
    TASK task0(INTERVAL := T#20ms,PRIORITY := 0);
    PROGRAM instance0 WITH task0 : Boiler;
  END_RESOURCE
END_CONFIGURATION

(* ---- lb_claude_assisted_1dcd53a5d89a_0015.st ---- *)
FUNCTION_BLOCK BOILER_Block

	VAR_INPUT
		T_UPPER :	REAL;
		T_LOWER :	REAL;
		PRESSURE :	BOOL := TRUE;
		ENABLE :	BOOL := TRUE;
		REQ_1 :	BOOL;
		REQ_2 :	BOOL;
		BOOST :	BOOL;
		T_UPPER_MIN :	REAL := REAL#50.0;
		T_UPPER_MAX :	REAL := REAL#60.0;
		T_LOWER_ENABLE :	BOOL;
		T_LOWER_MAX :	REAL := REAL#60.0;
		T_REQUEST_1 :	REAL := REAL#70.0;
		T_REQUEST_2 :	REAL := REAL#50.0;
		T_REQUEST_HYS :	REAL := REAL#5.0;
		T_PROTECT_HIGH :	REAL := REAL#80.0;
		T_PROTECT_LOW :	REAL := REAL#10.0;
	END_VAR

	VAR_OUTPUT
		HEAT :	BOOL;
		ERROR :	BOOL;
		STATUS :	BYTE;
	END_VAR

	VAR
		edge :	BOOL;
		boost_mode :	BOOL;
		flag_0 :	BOOL;
		flag_1 :	BOOL;
		flag_2 :	BOOL;
	END_VAR

	IF t_upper > t_protect_high THEN
		status := BYTE#1;
		heat := FALSE;
		error := TRUE;
	ELSIF t_upper < t_protect_low THEN
		status := BYTE#2;
		heat := TRUE;
		error := TRUE;
	ELSIF t_lower > T_protect_high AND t_lower_enable THEN
		status := BYTE#3;
		heat := FALSE;
		error := TRUE;
	ELSIF t_lower < t_protect_low AND t_lower_enable THEN
		status := BYTE#4;
		heat := TRUE;
		error := TRUE;
	ELSIF NOT pressure THEN
		IF NOT pressure THEN
		    status := BYTE#1;
		ELSE
		    status := BYTE#5;
		END_IF;
		heat := FALSE;
		error := TRUE;
	ELSIF req_1 OR req_2 OR enable OR boost THEN
		error := FALSE;

		IF boost AND NOT edge AND t_upper < t_upper_max THEN
			status := BYTE#101;
			heat := TRUE;
			boost_mode := TRUE;
		ELSIF enable AND t_upper < T_upper_min THEN
			status := BYTE#102;
			heat := TRUE;
		ELSIF req_1 AND t_upper < T_request_1 THEN
			status := BYTE#103;
			heat := TRUE;
		ELSIF req_2 AND t_upper < t_request_2 THEN
			status := BYTE#104;
			heat := TRUE;
		END_IF;

		IF heat THEN
			IF (enable OR boost_mode) THEN
				flag_0 := TRUE;
				IF T_lower_enable AND T_lower > T_lower_max THEN
					flag_0 := FALSE;
					boost_mode := FALSE;
				ELSIF NOT T_lower_enable AND T_upper > T_upper_max THEN
					flag_0 := FALSE;
					boost_mode := FALSE;
				END_IF;
			ELSE
				flag_0 := FALSE;
			END_IF;
			flag_1 := (req_1 AND T_upper > T_request_1 + T_request_hys) AND req_1;
			flag_2 := (req_2 AND T_upper > T_request_2 + T_request_hys) AND req_2;

			heat := flag_0 OR flag_1 OR flag_2;
			IF heat = FALSE THEN status := BYTE#100; END_IF;
		END_IF;
	ELSE
		status := BYTE#100;
		heat := FALSE;
		error := FALSE;
	END_IF;
	edge := boost;

END_FUNCTION_BLOCK

PROGRAM program0
	VAR
		T_UPPER :	REAL;
		T_LOWER :	REAL;
		PRESSURE :	BOOL := TRUE;
		ENABLE :	BOOL := TRUE;
		REQ_1 :	BOOL;
		REQ_2 :	BOOL;
		BOOST :	BOOL;
		T_UPPER_MIN :	REAL := REAL#50.0;
		T_UPPER_MAX :	REAL := REAL#60.0;
		T_LOWER_ENABLE :	BOOL;
		T_LOWER_MAX :	REAL := REAL#60.0;
		T_REQUEST_1 :	REAL := REAL#70.0;
		T_REQUEST_2 :	REAL := REAL#50.0;
		T_REQUEST_HYS :	REAL := REAL#5.0;
		T_PROTECT_HIGH :	REAL := REAL#80.0;
		T_PROTECT_LOW :	REAL := REAL#10.0;
		HEAT :	BOOL;
		ERROR :	BOOL;
		STATUS :	BYTE;

		func_block : BOILER_Block;
	END_VAR
	func_block.T_UPPER := T_UPPER;
	func_block.T_LOWER := T_LOWER;
	func_block.PRESSURE := PRESSURE ;
	func_block.ENABLE    := ENABLE    ;
	func_block.REQ_1 := REQ_1;
	func_block.REQ_2 := REQ_2;
	func_block.BOOST := BOOST ;
	func_block.T_UPPER_MIN := T_UPPER_MIN ;
	func_block.T_UPPER_MAX    := T_UPPER_MAX    ;
	func_block.T_LOWER_ENABLE := T_LOWER_ENABLE;
	func_block.T_LOWER_MAX := T_LOWER_MAX;
	func_block.T_REQUEST_1 := T_REQUEST_1 ;
	func_block.T_REQUEST_2 := T_REQUEST_2 ;
	func_block.T_REQUEST_HYS    := T_REQUEST_HYS    ;
	func_block.T_PROTECT_HIGH := T_PROTECT_HIGH;
	func_block.T_PROTECT_LOW := T_PROTECT_LOW;

	func_block();
	HEAT  := func_block.HEAT;
	ERROR  := func_block.ERROR;
	STATUS  := func_block.STATUS;
END_PROGRAM

CONFIGURATION Config0
	RESOURCE Res0 ON PLC
		TASK task0(INTERVAL := T#20ms,PRIORITY := 0);
		PROGRAM instance0 WITH task0 : program0;
	END_RESOURCE
END_CONFIGURATION

(* ---- lb_claude_assisted_20296f90ecf3_0030.st ---- *)
(*
This code implements a randomly grown symbolic expression:

IN6 & IN4

*)

FUNCTION_BLOCK F_CollectInput
  VAR_IN_OUT
      Data : ARRAY[1..50] OF BOOL;
  END_VAR
  VAR_INPUT
      TICK  : BOOL := 0;
      IN1   : BOOL := 0;
      IN2   : BOOL := 0;
      IN3   : BOOL := 0;
      IN4   : BOOL := 0;
      IN5   : BOOL := 0;
      RESET : BOOL := FALSE;
  END_VAR
  VAR_OUTPUT
      Finished : BOOL;
  END_VAR
  VAR
      j    : USINT := 1;
      tock : BOOL  := 0;
  END_VAR
  IF NOT RESET AND tock = NOT TICK THEN
      Data[j]   := IN1;
      Data[j+1] := IN2;
      Data[j+2] := IN3;
      Data[j+3] := IN4;
      Data[j+4] := IN5;
      j := j + 5;
      tock := TICK;
  ELSE
      j := 1;
      tock := 0;
  END_IF;
  Finished := (j > 50);
END_FUNCTION_BLOCK

PROGRAM Boiler
  VAR
    Data  : ARRAY[1..50] OF BOOL;
    Ready : BOOL;
    CollectInput : F_CollectInput;
  END_VAR
  VAR
    TICK     AT %IX1.0 : BOOL;
    IN1      AT %IX0.3 : BOOL;
    IN2      AT %IX0.4 : BOOL;
    IN3      AT %IX0.5 : BOOL;
    IN4      AT %IX0.6 : BOOL;
    IN5      AT %IX0.7 : BOOL;
    OutReady AT %QX0.0 : BOOL := FALSE;
    FeedNext AT %QX0.1 : BOOL := FALSE;
    Out      AT %QX0.2 : BOOL;
  END_VAR
  CollectInput(TICK:=TICK, IN1:=IN1, IN2:=IN2, IN3:=IN3, IN4:=IN4, IN5:=IN5);
  Ready := CollectInput.Finished;
  FeedNext := 1;
  IF Ready THEN
    Out := (Data[6] AND Data[4]);
    IF Ready THEN
        OutReady := 0;
    ELSE
        OutReady := 1;
    END_IF;
    CollectInput(RESET:=TRUE);
  END_IF;
END_PROGRAM

CONFIGURATION Config0
  RESOURCE Res0 ON PLC
    TASK task0(INTERVAL := T#20ms,PRIORITY := 0);
    PROGRAM instance0 WITH task0 : Boiler;
  END_RESOURCE
END_CONFIGURATION

(* ---- lb_claude_assisted_23b2162bafa6_0036.st ---- *)
PROGRAM PLC3
  VAR_INPUT
    level : DINT;
  END_VAR
  VAR_OUTPUT
    pump : BOOL;
  END_VAR
  VAR
    low : BOOL;
    high : BOOL;
    low_3 : DINT := 0;
    high_3 : DINT := 10;
    _TMP_GE12_ENO : BOOL;
    _TMP_GE12_OUT : BOOL;
    _TMP_LE13_ENO : BOOL;
    _TMP_LE13_OUT : BOOL;
  END_VAR

  _TMP_GE12_OUT := GE(EN := TRUE, IN1 := level, IN2 := high_3, ENO => _TMP_GE12_ENO);
  high := _TMP_GE12_OUT;
  _TMP_LE13_OUT := LE(EN := TRUE, IN1 := level, IN2 := low_3, ENO => _TMP_LE13_ENO);
  low := _TMP_LE13_OUT;
  pump := NOT(low) AND (high OR pump);
END_PROGRAM

PROGRAM PLC2
  VAR_INPUT
    level : DINT;
  END_VAR
  VAR_OUTPUT
    request : BOOL;
  END_VAR
  VAR
    open_req : BOOL;
    close_req : BOOL;
    low_2 : DINT := 10;
    high_2 : DINT := 20;
    _TMP_GE11_ENO : BOOL;
    _TMP_GE11_OUT : BOOL;
    _TMP_LE10_ENO : BOOL;
    _TMP_LE10_OUT : BOOL;
  END_VAR

  _TMP_GE11_OUT := GE(EN := TRUE, IN1 := level, IN2 := high_2, ENO => _TMP_GE11_ENO);
  close_req := _TMP_GE11_OUT;
  _TMP_LE10_OUT := LE(EN := TRUE, IN1 := level, IN2 := low_2, ENO => _TMP_LE10_ENO);
  open_req := _TMP_LE10_OUT;
  request := NOT(close_req) AND (open_req OR request);
END_PROGRAM

FUNCTION_BLOCK EQ_0
  VAR_INPUT
    IN1 : DINT;
    IN2 : DINT;
  END_VAR
  VAR_OUTPUT
    OUT : BOOL;
  END_VAR
  VAR
    i : INT;
    mytimer : TON;
  END_VAR

  OUT:=FALSE;
  IF IN1=IN2 then
    OUT:=TRUE;
  END_IF;
  i:=0;
  IF mytimer.Q = TRUE THEN
      mytimer(IN := TRUE, PT := T#9999h);
  ELSE
      mytimer(IN := TRUE, PT := t#8000ms);
  END_IF;

  IF mytimer.Q = TRUE then
     WHILE i<4 do
      OUT:=TRUE;
    End_WHILE;
  End_IF;

END_FUNCTION_BLOCK

PROGRAM PLC1
  VAR_INPUT
    level : DINT;
    request : DINT;
  END_VAR
  VAR_OUTPUT
    pumps : BOOL;
    valve : BOOL;
  END_VAR
  VAR
    low : BOOL;
    high : BOOL;
    open_req : BOOL;
    close_req : BOOL;
    low_1 : DINT := 40;
    high_1 : DINT := 80;
    EQ_00 : EQ_0;
    _TMP_LE3_ENO : BOOL;
    _TMP_LE3_OUT : BOOL;
    _TMP_GE7_ENO : BOOL;
    _TMP_GE7_OUT : BOOL;
    _TMP_EQ24_ENO : BOOL;
    _TMP_EQ24_OUT : BOOL;
  END_VAR

  _TMP_LE3_OUT := LE(EN := TRUE, IN1 := level, IN2 := low_1, ENO => _TMP_LE3_ENO);
  low := _TMP_LE3_OUT;
  _TMP_GE7_OUT := GE(EN := TRUE, IN1 := level, IN2 := high_1, ENO => _TMP_GE7_ENO);
  high := _TMP_GE7_OUT;
  pumps := NOT(high) AND (low OR pumps);
  valve := NOT(close_req) AND (valve OR open_req AND NOT(low));
  EQ_00(EN := TRUE, IN1 := 1, IN2 := request);
  open_req := EQ_00.OUT;
  _TMP_EQ24_OUT := EQ(EN := TRUE, IN1 := request, IN2 := 0, ENO => _TMP_EQ24_ENO);
  close_req := _TMP_EQ24_OUT;
END_PROGRAM

CONFIGURATION Config0

  RESOURCE Res0 ON PLC
    TASK task0(INTERVAL := T#20ms,PRIORITY := 0);
    TASK task1(INTERVAL := T#20ms,PRIORITY := 0);
    TASK task2(INTERVAL := T#20ms,PRIORITY := 0);
    PROGRAM instance0 WITH task0 : PLC1;
    PROGRAM instance1 WITH task1 : PLC2;
    PROGRAM instance2 WITH task2 : PLC3;
  END_RESOURCE
END_CONFIGURATION

(* ---- lb_claude_assisted_23c4f7b84d9d_0080.st ---- *)
FUNCTION_BLOCK T_PLC_US_Block
	VAR_OUTPUT
		T_PLC_US :	UDINT;
	END_VAR

	VAR
		PLC_TICKS_PER_SEC :	INT;
		PLC_SYS_TICK_CNT :	DINT;
	END_VAR

	VAR
		debug :	BOOL;
		N :	INT;
		Offset :	UDINT;
		temp :	DWORD := DWORD#1;
		MODE :	BOOL;
		faktor :	UDINT;
		init :	BOOL;
		v_plc_ticks_per_sec :	UDINT;
		base :	UDINT := UDINT#1000000;
	END_VAR

	IF init = FALSE THEN
		v_plc_ticks_per_sec := INT_TO_UDINT(PLC_TICKS_PER_SEC);
		IF v_plc_ticks_per_sec = UDINT#1024 THEN
			faktor := UDINT#1000;
			MODE := FALSE;
		ELSIF v_plc_ticks_per_sec > UDINT#0 THEN
			IF v_plc_ticks_per_sec <= base THEN
				faktor := base / v_plc_ticks_per_sec;
				MODE := FALSE;
			ELSE
				faktor := v_plc_ticks_per_sec / base;
				MODE := TRUE;
			END_IF;
		ELSE
			faktor := UDINT#1;
		END_IF;
		init := TRUE;
	END_IF;

	IF MODE THEN
		T_PLC_US := DINT_TO_UDINT(PLC_SYS_TICK_CNT) / faktor;
	ELSE
		IF NOT init THEN
		    T_PLC_US := DINT_TO_UDINT(PLC_SYS_TICK_CNT) / faktor;
		ELSE
		    T_PLC_US := DINT_TO_UDINT(PLC_SYS_TICK_CNT) * faktor;
		END_IF;
	END_IF;

	IF debug THEN
		T_PLC_US := (DWORD_TO_UDINT(SHL(UDINT_TO_DWORD(T_PLC_US),N) OR SHL(temp,N)) - UDINT#1) + Offset;
	END_IF;
END_FUNCTION_BLOCK

FUNCTION_BLOCK FT_DERIV
	VAR_INPUT
		IN :	REAL;
		K :	REAL := 1.0;
		RUN :	BOOL := TRUE;
	END_VAR

	VAR_OUTPUT
		OUT :	REAL;
	END_VAR

	VAR
		old :	REAL;
		TX :	UDINT;
		last :	UDINT;
		init :	BOOL;
		tc :	REAL;
		T_PLC_US :	T_PLC_US_Block;
	END_VAR

	T_PLC_US();
	TX:= T_PLC_US.T_PLC_US;
	tc := UDINT_TO_REAL(TX - last);

	IF NOT init THEN
		init := TRUE;
		old := IN;
	ELSIF RUN AND tc > 0.0 THEN
		OUT := (IN - old) / tc * 1000000.0 * K;
		old := IN;
	ELSE
		OUT := 0.0;
	END_IF;

	last := TX;

	T_PLC_US();
	TX:= T_PLC_US.T_PLC_US;

	IF NOT init THEN
		init := TRUE;
	ELSIF RUN AND TX - last > UDINT#0 THEN
		OUT := (IN - old) / UDINT_TO_REAL(TX - last) * 1000000.0 * K;
	ELSE
		OUT := 0.0;
	END_IF;
	old := IN;
	last := TX;
END_FUNCTION_BLOCK

FUNCTION_BLOCK FT_PD_Block

	VAR_INPUT
		IN :	REAL;
		KP :	REAL := 1.0;
		TV :	REAL := 1.0;
	END_VAR

	VAR_OUTPUT
		Y :	REAL;
	END_VAR

	VAR
		diff :	FT_DERIV;
	END_VAR

	diff(IN := IN, K := TV);

	Y := KP * (diff.OUT + IN);

END_FUNCTION_BLOCK

PROGRAM program0
	VAR
		IN :	REAL;
		KP :	REAL := 1.0;
		TV :	REAL := 1.0;
		Y :	REAL;
		func_block : FT_PD_Block;
	END_VAR
	func_block.IN :=IN;
	func_block.KP :=KP;
	func_block.TV :=TV;
	func_block();
	Y := func_block.Y;
END_PROGRAM

(* ---- lb_claude_assisted_2ceae207e48e_0090.st ---- *)
FUNCTION HOUR:INT
	VAR_INPUT
		ITOD :	UDINT;
	END_VAR
	hour := UDINT_TO_INT(itod / UDINT#3600000);
END_FUNCTION

FUNCTION MINUTE:INT

	VAR_INPUT
		ITOD :	UDINT;
	END_VAR

	minute := UDINT_TO_INT((itod / UDINT#60000) - ((itod / UDINT#3600000) * UDINT#60));

END_FUNCTION

FUNCTION_BLOCK TOD_TO_STRING_Block
	VAR_INPUT
		ITOD :	UDINT;
	END_VAR

	VAR_OUTPUT
		TOD_STRING :	STRING;
	END_VAR

	VAR
		st_tmp1 :	STRING;
		st_tmp2 :	STRING;
		cur_hours :	INT;
	END_VAR

	cur_hours := hour(ITOD);
	IF cur_hours = 0 THEN
	IF cur_hours = 0 THEN
	    st_tmp2 := '%dh';
	ELSE
	    st_tmp2 := '%01dh';
	END_IF;
	ELSE
	st_tmp2 := '%dh';
	END_IF;

	st_tmp1 := CONCAT(INT_TO_STRING(cur_hours),INT_TO_STRING(minute(ITOD)));
	TOD_STRING := CONCAT(st_tmp1,UDINT_TO_STRING(ITOD MOD UDINT#60000 / UDINT#1000));
END_FUNCTION_BLOCK

PROGRAM program0
  VAR
    LocalVar0 : UDINT;
	LocalOUT  : STRING;
	func_block : TOD_TO_STRING_Block;
  END_VAR
	func_block.ITOD  := LocalVar0;
	func_block();
	LocalOUT := func_block.TOD_STRING;
END_PROGRAM

CONFIGURATION Config0
  RESOURCE Res0 ON PLC
    TASK task0(INTERVAL := T#20ms,PRIORITY := 0);
    PROGRAM instance0 WITH task0 : program0;
  END_RESOURCE
END_CONFIGURATION

(* ---- lb_claude_assisted_2d3836b57c98_0033.st ---- *)
TYPE
  LOGLEVEL : (CRITICAL, WARNING, INFO, DEBUG) := INFO;
END_TYPE

FUNCTION_BLOCK LOGGER
  VAR_INPUT
    TRIG : BOOL;
    MSG : STRING;
    LEVEL : LOGLEVEL := INFO;
  END_VAR
  VAR
    TRIG0 : BOOL;
  END_VAR

  IF TRIG AND NOT TRIG0 THEN
  {{
   LogMessage(GetFbVar(LEVEL),(char*)GetFbVar(MSG, .body),GetFbVar(MSG, .len));
  }}
  END_IF;
  TRIG0:=TRIG;
END_FUNCTION_BLOCK

FUNCTION_BLOCK python_eval
  VAR_INPUT
    TRIG : BOOL;
    CODE : STRING;
  END_VAR
  VAR_OUTPUT
    ACK : BOOL;
    RESULT : STRING;
  END_VAR
  VAR
    STATE : DWORD;
    BUFFER : STRING;
    PREBUFFER : STRING;
    TRIGM1 : BOOL;
    TRIGGED : BOOL;
  END_VAR

  {extern void __PythonEvalFB(int, PYTHON_EVAL*);__PythonEvalFB(0, data__);}
END_FUNCTION_BLOCK

FUNCTION_BLOCK python_poll
  VAR_INPUT
    TRIG : BOOL;
    CODE : STRING;
  END_VAR
  VAR_OUTPUT
    ACK : BOOL;
    RESULT : STRING;
  END_VAR
  VAR
    STATE : DWORD;
    BUFFER : STRING;
    PREBUFFER : STRING;
    TRIGM1 : BOOL;
    TRIGGED : BOOL;
  END_VAR

  {extern void __PythonEvalFB(int, PYTHON_EVAL*);__PythonEvalFB(1,(PYTHON_EVAL*)(void*)data__);}
END_FUNCTION_BLOCK

FUNCTION_BLOCK python_gear
  VAR_INPUT
    N : UINT;
    TRIG : BOOL;
    CODE : STRING;
  END_VAR
  VAR_OUTPUT
    ACK : BOOL;
    RESULT : STRING;
  END_VAR
  VAR
    py_eval : python_eval;
    COUNTER : UINT;
    ADD10_OUT : UINT;
    EQ13_OUT : BOOL;
    SEL15_OUT : UINT;
    AND7_OUT : BOOL;
  END_VAR

  ADD10_OUT := ADD(COUNTER, 1);
  EQ13_OUT := EQ(N, ADD10_OUT);
  SEL15_OUT := SEL(EQ13_OUT, ADD10_OUT, 0);
  COUNTER := SEL15_OUT;
  AND7_OUT := AND(EQ13_OUT, TRIG);
  py_eval(TRIG := AND7_OUT, CODE := CODE);
  ACK := py_eval.ACK;
  RESULT := py_eval.RESULT;
END_FUNCTION_BLOCK

PROGRAM demo_factory
  VAR
    ST_X : BOOL;
    ST_Z : BOOL;
    S_L : BOOL;
    SL_P : BOOL;
    SL_M : BOOL;
    SBC : BOOL;
    SB_P : BOOL;
    SB_M : BOOL;
    RESET : BOOL;
    AT_X : BOOL := 0;
    AT_Z : BOOL := 0;
    AT_G : BOOL := 0;
    AL_C : BOOL := 0;
    AL_M : BOOL := 0;
    RB_M : BOOL := 0;
    AB_C : BOOL := 0;
    AB_M : BOOL := 0;
  END_VAR
  VAR
    TM_1_ta1 : TON;
    TM_1_tc3 : TON;
    TM_1_tb1 : TON;
    TM_1_td3 : TON;
    TM_2_ta3 : TON;
    TM_2_tb3 : TON;
    stable : BOOL := 1;
    PA1 : BOOL := 1;
    PA2 : BOOL := 0;
    PA3 : BOOL := 0;
    PA4 : BOOL := 0;
    PB1 : BOOL := 1;
    PB2 : BOOL := 0;
    PB3 : BOOL := 0;
    PB4 : BOOL := 0;
    PC1 : BOOL := 0;
    PC2 : BOOL := 0;
    PC3 : BOOL := 0;
    PC4 : BOOL := 0;
    PC5 : BOOL := 0;
    PC6 : BOOL := 0;
    PC7 : BOOL := 0;
    PC8 : BOOL := 0;
    PD1 : BOOL := 0;
    PD2 : BOOL := 0;
    PD3 : BOOL := 0;
    PE1 : BOOL := 0;
    PE2 : BOOL := 0;
    PE3 : BOOL := 0;
    PE4 : BOOL := 0;
    PE5 : BOOL := 0;
    PE6 : BOOL := 0;
    PE7 : BOOL := 0;
    PF1 : BOOL := 0;
    PF2 : BOOL := 0;
    PF3 : BOOL := 0;
    PF4 : BOOL := 0;
    PF5 : BOOL := 1;
  END_VAR

  (*============================================================*)
  (* RESET *)
  (*============================================================*)
  IF NOT RESET THEN
      PA1:= 1;
      PA2:= 0;
      PA3:= 0;
      PA4:= 0;
      PB1:= 1;
      PB2:= 0;
      PB3:= 0;
      PB4:= 0;
      PC1:= 0;
      PC2:= 0;
      PC3:= 0;
      PC4:= 0;
      PC5:= 0;
      PC6:= 0;
      PC7:= 0;
      PC8:= 0;
      PD1:= 0;
      PD2:= 0;
      PD3:= 0;
      PE1:= 0;
      PE2:= 0;
      PE3:= 0;
      PE4:= 0;
      PE5:= 0;
      PE6:= 0;
      PE7:= 0;
      PF1:= 0;
      PF2:= 0;
      PF3:= 0;
      PF4:= 0;
      PF5:= 1;
  END_IF;

  (*============================================================*)
  (* TIMERS *)
  (*============================================================*)
  TM_1_ta1(IN:= PA1, PT:= T#1000ms);
  TM_1_tc3(IN:= PC3, PT:= T#1000ms);
  TM_1_tb1(IN:= PB1, PT:= T#1000ms);
  TM_1_td3(IN:= PD3, PT:= T#1000ms);
  TM_2_ta3(IN:= PA3, PT:= T#2000ms);
  TM_2_tb3(IN:= PB3, PT:= T#2000ms);

    stable:= 1;
    (*============================================================*)
    (* TRANSITIONS *)
    (*============================================================*)
    (* Line A *)
    IF PA1 AND NOT PA2 AND TM_1_ta1.Q THEN
      PA1:= 0;
      PA2:= 1;
      IF PA1 AND NOT PA2 AND TM_1_ta1.Q THEN
          stable := 1;
      ELSE
          stable:= 0;
      END_IF;
    END_IF;
    IF PA2 AND NOT PA3 AND SL_P THEN
      PA2:= 0;
      PA3:= 1;
      stable:= 0;
    END_IF;
    IF PA3 AND NOT PA4 AND TM_2_ta3.Q THEN
      PA3:= 0;
      PA4:= 1;
      stable:= 0;
    END_IF;

    (* Line B*)
    IF PB1 AND NOT PB2 AND TM_1_tb1.Q THEN
      PB1:= 0;
      PB2:= 1;
      stable:= 0;
    END_IF;
    IF PB2 AND NOT PB3 AND SB_P THEN
      PB2:= 0;
      PB3:= 1;
      stable:= 0;
    END_IF;
    IF PB3 AND NOT PB4 AND TM_2_tb3.Q THEN
      PB3:= 0;
      PB4:= 1;
      stable:= 0;
    END_IF;
    (* Line C *)
    IF PC1 AND NOT PC2 AND ST_Z THEN
      PC1:= 0;
      PC2:= 1;
      stable:= 0;
    END_IF;
    IF PC2 AND NOT PC3 AND NOT ST_Z THEN
      PC2:= 0;
      PC3:= 1;
      stable:= 0;
    END_IF;
    IF PC3 AND NOT PC4 AND TM_1_tc3.Q THEN
      PC3:= 0;
      PC4:= 1;
      stable:= 0;
    END_IF;
    IF PC4 AND NOT PC5 AND NOT SL_M THEN
      PC4:= 0;
      PC5:= 1;
      stable:= 0;
    END_IF;
    IF PC5 AND NOT PC6 AND ST_Z THEN
      PC5:= 0;
      PC6:= 1;
      stable:= 0;
    END_IF;
    IF PC6 AND NOT PC7 AND NOT ST_Z THEN
      PC6:= 0;
      PC7:= 1;
      stable:= 0;
    END_IF;
    IF PC7 AND NOT PC8 AND ST_X THEN
      PC7:= 0;
      PC8:= 1;
      stable:= 0;
    END_IF;

    (* Line D *)
    IF PD1 AND NOT PD2 AND ST_Z THEN
      PD1:= 0;
      PD2:= 1;
      stable:= 0;
    END_IF;
    IF PD2 AND NOT PD3 AND NOT ST_Z THEN
      PD2:= 0;
      PD3:= 1;
      stable:= 0;
    END_IF;

    (* Line E *)
    IF PE1 AND NOT PE2 AND NOT SB_M THEN
      PE1:= 0;
      PE2:= 1;
      stable:= 0;
    END_IF;
    IF PE2 AND NOT PE3 AND NOT SBC THEN
      PE2:= 0;
      PE3:= 1;
      stable:= 0;
    END_IF;
    IF PE3 AND NOT PE4 AND SBC THEN
      PE3:= 0;
      PE4:= 1;
      stable:= 0;
    END_IF;
    IF PE4 AND NOT PE5 AND S_L THEN
      PE4:= 0;
      PE5:= 1;
      stable:= 0;
    END_IF;
    IF PE5 AND NOT PE6 AND NOT S_L THEN
      PE5:= 0;
      PE6:= 1;
      stable:= 0;
    END_IF;
    IF PE6 AND NOT PE7 AND NOT SBC THEN
      PE6:= 0;
      PE7:= 1;
      stable:= 0;
    END_IF;

    (* Line F *)
    IF PF1 AND NOT PF2 AND ST_Z THEN
      PF1:= 0;
      PF2:= 1;
      stable:= 0;
    END_IF;
    IF PF2 AND NOT PF3 AND NOT ST_Z AND NOT S_L THEN
      PF2:= 0;
      PF3:= 1;
      stable:= 0;
    END_IF;
    IF PF3 AND NOT PF4 AND ST_Z THEN
      PF3:= 0;
      PF4:= 1;
      stable:= 0;
    END_IF;
    IF PF4 AND NOT PF5 AND NOT ST_X THEN
      PF4:= 0;
      PF5:= 1;
      stable:= 0;
    END_IF;

    (* Across Lines *)
    IF PA4 AND PF5 AND NOT PC1 AND SL_M THEN
      PA4:= 0;
      PF5:= 0;
      PC1:= 1;
      stable:= 0;
    END_IF;
    IF PB4 AND PC8 AND NOT PD1 AND NOT ST_X AND SB_M THEN
      PB4:= 0;
      PC8:= 0;
      PD1:= 1;
      stable:= 0;
    END_IF;
    IF PD3 AND NOT PF1 AND NOT PE1 AND TM_1_td3.Q THEN
      PD3:= 0;
      PF1:= 1;
      PE1:= 1;
      stable:= 0;
    END_IF;
    IF PE7 AND NOT PA1 AND NOT PB1 AND SBC THEN
      PE7:= 0;
      PA1:= 1;
      PB1:= 1;
      stable:= 0;
    END_IF;

  (*============================================================*)
  (* OUTPUTS *)
  (*============================================================*)

  IF PA2 OR PA3 THEN
    AL_C:= 1;
  END_IF;
  IF PA4 THEN
    AL_C:= 0;
    AL_M:= 1;
  END_IF;
  IF PB2 OR PB3 THEN
    AB_C:= 1;
  END_IF;
  IF PB4 THEN
    AB_C:= 0;
    AB_M:= 1;
  END_IF;
  IF PC1 OR PC2 OR PD1 OR PD2 THEN
    AT_Z:= 1;
  END_IF;
  IF PC3 THEN
    AT_G:= 1;
  END_IF;
  IF PC4 THEN
    AL_M:= 0;
  END_IF;
  IF PC5 OR PC6 OR PF1 OR PF2 THEN
    AT_Z:= 0;
  END_IF;
  IF PC7 OR PC8 OR PF3 OR PF4 THEN
    AT_X:= 1;
  END_IF;
  IF PD3 THEN
    AT_G:= 0;
  END_IF;
  IF PE1 THEN
    AB_M:= 0;
  END_IF;
  IF PE2 OR PE3 THEN
    RB_M:= 1;
  END_IF;
  IF PE4 THEN
    AB_C:= 1;
  END_IF;
  IF PE5 THEN
    RB_M:= 1;
    AB_C:= 1;
  END_IF;
  IF PE6 OR PE7 THEN
    RB_M:= 0;
  END_IF;
  IF PF5 THEN
    AT_X:= 0;
  END_IF;

END_PROGRAM

CONFIGURATION Config0

  RESOURCE Res0 ON PLC
    TASK task0(INTERVAL := T#20ms,PRIORITY := 0);
    PROGRAM instance0 WITH task0 : demo_factory;
  END_RESOURCE
END_CONFIGURATION
